KUKA KRL program: UP24.src, Up24.dat

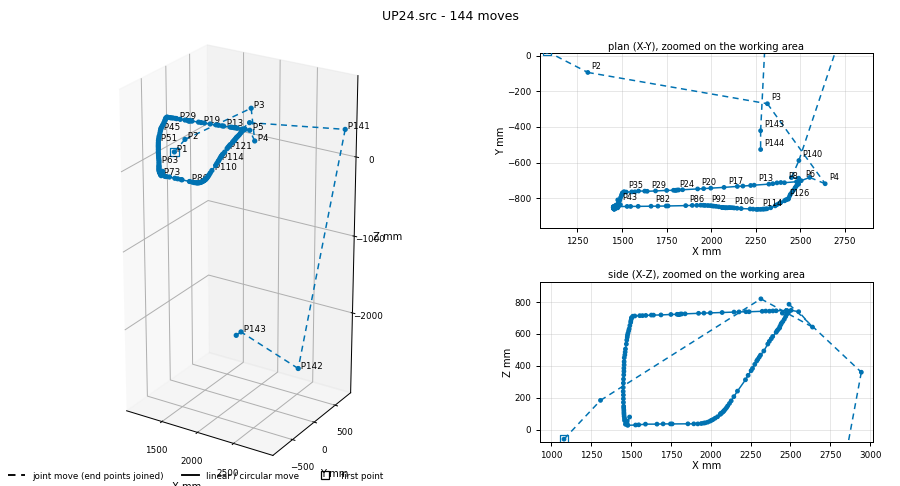
[picture p0: tool path of UP24.src, 144 of 144 moves have a stored position in this frame; points joined in program order, loops and branches not executed]
--- UP24.src ---
&ACCESS RVO1
&REL 1255
&COMMENT VW380 Klebeauftrag_AFO415600
&PARAM EDITMASK = Up999[1-999]
&PARAM TEMPLATE = C:\KRC\Roboter\Template\upvorgabe
&PARAM TPVW_VERSION = 8.3.18
&PARAM DISKPATH = KRC:\R1\UPs
DEF UP24()
   ; FOLD UP Anfang;%{SE} %MKUKATPVW
   SPS_N=-1
   SPS_FERTIG=FALSE
   IF NOT CALLBYSELECT THEN
      INTERRUPT DECL 10 WHEN $CYCFLAG[254]==FALSE DO VW(#FB_STOP,TRUE)
      INTERRUPT ON 10
      INT10=TRUE
      VW_USR_R (#USR_INIT)
   ENDIF
   VW(#VW_INIT_UP,TRUE)
   ; ENDFOLD
   ;FOLD -- VW380, THIL -- ;%{PSE}%MKUKATPVW,%CVW_COM,%VCOMMENT,%P 1:Comment:, 2:VW380, THIL
      ;FOLD {H}
         M_COMMENT("VW380, THIL")
      ;ENDFOLD
   ;ENDFOLD
   ;FOLD -- 415600R01 -- ;%{PSE}%MKUKATPVW,%CVW_COM,%VCOMMENT,%P 1:Comment:, 2:415600R01
      ;FOLD {H}
         M_COMMENT("415600R01")
      ;ENDFOLD
   ;ENDFOLD
   ;FOLD -- FRG ST415600 -- ;%{PSE}%MKUKATPVW,%CVW_COM,%VCOMMENT,%P 1:Comment:, 2:FRG ST415600
      ;FOLD {H}
         M_COMMENT("FRG ST415600")
      ;ENDFOLD
   ;ENDFOLD
   ;FOLD -- ACHTUNG! Position ist nicht von PF0 anfahrbar! -- ;%{PSE}%MKUKATPVW,%CVW_COM,%VCOMMENT,%P 1:Comment:, 2:ACHTUNG! Position ist nicht von PF0 anfahrbar!
      ;FOLD {H}
         M_COMMENT("ACHTUNG! Position ist nicht von PF0 anfahrbar!")
      ;ENDFOLD
   ;ENDFOLD
   ;FOLD PTP VB=100% VE=0% ACC=100% RobWzg=1 Base=2 SPSTrig=0[1/100s] P ;%{P}%MKUKATPVW,%CMOVE8,%VPTP,%P 1:1, 2: VB=, 3:100, 4:%, 5: VE=, 6:0, 7:%, 8: ACC=, 9:100, 10:%, 11: RobWzg=, 12:1, 13: Base=, 14:2, 15: SPSTrig=, 16:0, 17:[1/100s], 18: P, 19:1, 20:-1, 21:200001
      ;FOLD 1: FB PSPS = EIN ;%{SE}%MKUKATPVW %CVW_SPS %VFBPSPS %P 2:FB PSPS = EIN,3:FBPSPS
      ;ENDFOLD
      ;FOLD 2: t5 ( EIN ) = 0[1/10Sek] ;%{SE}%MKUKATPVW %CVW_SPS %VTASG %P 2:t5 ( EIN ) = 0[1/10Sek],3:TASG
      ;ENDFOLD
      ;FOLD 3: A23 = AUS ;%{SE}%MKUKATPVW %CVW_SPS %VBOASG %P 2:A23 = AUS,3:BOASG
      ;ENDFOLD
      ;FOLD 4: SPSMAKRO50 = EIN ;%{SE}%MKUKATPVW %CVW_SPS %VMAKRO %P 2:SPSMAKRO50 = EIN,3:MAKRO
      ;ENDFOLD
      ;FOLD 5: A65 = AUS ;%{SE}%MKUKATPVW %CVW_SPS %VBOASG %P 2:A65 = AUS,3:BOASG
      ;ENDFOLD
      ;FOLD 6: A68 = EIN ;%{SE}%MKUKATPVW %CVW_SPS %VBOASG %P 2:A68 = EIN,3:BOASG
      ;ENDFOLD
      ;FOLD 7: A69 = AUS ;%{SE}%MKUKATPVW %CVW_SPS %VBOASG %P 2:A69 = AUS,3:BOASG
      ;ENDFOLD
      ;FOLD 8: A71 = AUS ;%{SE}%MKUKATPVW %CVW_SPS %VBOASG %P 2:A71 = AUS,3:BOASG
      ;ENDFOLD
      ;FOLD 9: A72 = EIN ;%{SE}%MKUKATPVW %CVW_SPS %VBOASG %P 2:A72 = EIN,3:BOASG
      ;ENDFOLD
      ;FOLD 10: A73 = AUS ;%{SE}%MKUKATPVW %CVW_SPS %VBOASG %P 2:A73 = AUS,3:BOASG
      ;ENDFOLD
      ;FOLD 11: A76 = EIN ;%{SE}%MKUKATPVW %CVW_SPS %VBOASG %P 2:A76 = EIN,3:BOASG
      ;ENDFOLD
      ;FOLD 12: A77 = AUS ;%{SE}%MKUKATPVW %CVW_SPS %VBOASG %P 2:A77 = AUS,3:BOASG
      ;ENDFOLD
      ;FOLD 13: A80 = EIN ;%{SE}%MKUKATPVW %CVW_SPS %VBOASG %P 2:A80 = EIN,3:BOASG
      ;ENDFOLD
      ;FOLD 14: F930 = AUS ;%{SE}%MKUKATPVW %CVW_SPS %VBOASG %P 2:F930 = AUS,3:BOASG
      ;ENDFOLD
      ;FOLD 15: F939 = AUS ;%{SE}%MKUKATPVW %CVW_SPS %VBOASG %P 2:F939 = AUS,3:BOASG
      ;ENDFOLD
      ;FOLD 16: F1 = EIN ;%{SE}%MKUKATPVW %CVW_SPS %VBOASG %P 2:F1 = EIN,3:BOASG
      ;ENDFOLD
      ;FOLD 17: SPSMAKRO343 = !M32 ;%{SE}%MKUKATPVW %CVW_SPS %VMAKRO %P 2:SPSMAKRO343 = !M32,3:MAKRO
      ;ENDFOLD
      ;FOLD 18: SPSMAKRO340 = EIN ;%{SE}%MKUKATPVW %CVW_SPS %VMAKRO %P 2:SPSMAKRO340 = EIN,3:MAKRO
      ;ENDFOLD
      ;FOLD 19: WARTE BIS M13 & M32 ;%{SE}%MKUKATPVW %CVW_SPS %VWBOASG %P 2:WARTE BIS M13 & M32,3:WBOASG
      ;ENDFOLD
      ;FOLD 20: A1521 = EIN ;%{SE}%MKUKATPVW %CVW_SPS %VBOASG %P 2:A1521 = EIN,3:BOASG
      ;ENDFOLD
      ;FOLD 21: A1522 = AUS ;%{SE}%MKUKATPVW %CVW_SPS %VBOASG %P 2:A1522 = AUS,3:BOASG
      ;ENDFOLD
      ;FOLD 22: A1523 = AUS ;%{SE}%MKUKATPVW %CVW_SPS %VBOASG %P 2:A1523 = AUS,3:BOASG
      ;ENDFOLD
      ;FOLD 23: WARTE BIS E1521 & !E1522 & !E1523 ;%{SE}%MKUKATPVW %CVW_SPS %VWBOASG %P 2:WARTE BIS E1521 & !E1522 & !E1523,3:WBOASG
      ;ENDFOLD
      ;FOLD 24: WARTE BIS M13 & M32 ;%{SE}%MKUKATPVW %CVW_SPS %VWBOASG %P 2:WARTE BIS M13 & M32,3:WBOASG
      ;ENDFOLD
      ;FOLD 25: bin10 ( EIN ) = 20 ;%{SE}%MKUKATPVW %CVW_SPS %VARIASG %P 2:bin10 ( EIN ) = 20,3:ARIASG
      ;ENDFOLD
      ;FOLD 26: bin11 ( EIN ) = 1 ;%{SE}%MKUKATPVW %CVW_SPS %VARIASG %P 2:bin11 ( EIN ) = 1,3:ARIASG
      ;ENDFOLD
      ;FOLD 27: F341 = EIN ;%{SE}%MKUKATPVW %CVW_SPS %VBOASG %P 2:F341 = EIN,3:BOASG
      ;ENDFOLD
      ;FOLD 28: ana1 ( EIN ) = VPROP: 500 [mm/Sek] OFFS: 0[mV] DELAY:0 [ms] ;%{SE}%MKUKATPVW %CVW_SPS %VANAVPROP %P 2:ana1 ( EIN ) = VPROP: 500 [mm/Sek] OFFS: 0[mV] DELAY:0 [ms],3:ANAVPROP
      ;ENDFOLD
      ;FOLD 29: A43 = AUS ;%{SE}%MKUKATPVW %CVW_SPS %VBOASG %P 2:A43 = AUS,3:BOASG
      ;ENDFOLD
      ;FOLD 30: A44 = AUS ;%{SE}%MKUKATPVW %CVW_SPS %VBOASG %P 2:A44 = AUS,3:BOASG
      ;ENDFOLD
      ;FOLD 31: WARTE BIS M32 & M34 & E43 & E44 & E63 & E71 ;%{SE}%MKUKATPVW %CVW_SPS %VWBOASG %P 2:WARTE BIS M32 & M34 & E43 & E44 & E63 & E71,3:WBOASG
      ;ENDFOLD
      ;FOLD 32: WARTE BIS E23 ;%{SE}%MKUKATPVW %CVW_SPS %VWBOASG %P 2:WARTE BIS E23,3:WBOASG
      ;ENDFOLD
      ;FOLD 33: A23 = EIN ;%{SE}%MKUKATPVW %CVW_SPS %VBOASG %P 2:A23 = EIN,3:BOASG
      ;ENDFOLD
      ;FOLD 34: FB PSPS = M13 & M30 & M32 & M34 & E43 & E44 & E63 & E71 ;%{SE}%MKUKATPVW %CVW_SPS %VFBPSPS %P 2:FB PSPS = M13 & M30 & M32 & M34 & E43 & E44 & E63 & E71,3:FBPSPS
      ;ENDFOLD
      ;FOLD {H}
         VW_MPARA_ACT=P1_D
         Act_P1 = P1
         Act_P2 = P1
         VW(#MPARA,TRUE)
         SPS_FERTIG=FALSE
         SPS_FERTIG_ANA=FALSE
         TRIGGER WHEN DISTANCE=1 DELAY=0 DO SPS_TRIG(1) PRIO=-1
         TRIGGER WHEN DISTANCE=1 DELAY=0 DO SPS_TRIG(20002) PRIO=-1
         PTP P1
         $ADVANCE=1
         WAIT FOR SPS_FERTIG
         WAIT FOR SPS_FERTIG_ANA
      ;ENDFOLD
   ;ENDFOLD
   ;FOLD PTP VB=100% VE=100% ACC=100% RobWzg=1 Base=2 SPSTrig=0[1/100s] P ;%{P}%MKUKATPVW,%CMOVE8,%VPTP,%P 1:1, 2: VB=, 3:100, 4:%, 5: VE=, 6:100, 7:%, 8: ACC=, 9:100, 10:%, 11: RobWzg=, 12:1, 13: Base=, 14:2, 15: SPSTrig=, 16:0, 17:[1/100s], 18: P, 19:2, 20:-1, 21:3
      ;FOLD 1: FB PSPS = M13 & M30 & M32 & M34 & E43 & E44 & E63 & E71 ;%{SE}%MKUKATPVW %CVW_SPS %VFBPSPS %P 2:FB PSPS = M13 & M30 & M32 & M34 & E43 & E44 & E63 & E71,3:FBPSPS
      ;ENDFOLD
      ;FOLD {H}
         VW_MPARA_ACT=P2_D
         Act_P1 = P2
         Act_P2 = P2
         VW(#MPARA,TRUE)
         SPS_FERTIG=FALSE
         TRIGGER WHEN DISTANCE=1 DELAY=0 DO SPS_TRIG(10003) PRIO=-1 UP_TIME_OUT=SPS_TIMEOUT
         PTP P2 C_PTP C_VEL
         $ADVANCE=1
      ;ENDFOLD
   ;ENDFOLD
   ;FOLD PTP VB=100% VE=100% ACC=100% RobWzg=1 Base=2 SPSTrig=0[1/100s] P ;%{P}%MKUKATPVW,%CMOVE8,%VPTP,%P 1:1, 2: VB=, 3:100, 4:%, 5: VE=, 6:100, 7:%, 8: ACC=, 9:100, 10:%, 11: RobWzg=, 12:1, 13: Base=, 14:2, 15: SPSTrig=, 16:0, 17:[1/100s], 18: P, 19:3, 20:-1, 21:4
      ;FOLD 1: FB PSPS = M13 & M30 & M32 & M34 & E43 & E44 & E63 & E71 ;%{SE}%MKUKATPVW %CVW_SPS %VFBPSPS %P 2:FB PSPS = M13 & M30 & M32 & M34 & E43 & E44 & E63 & E71,3:FBPSPS
      ;ENDFOLD
      ;FOLD {H}
         VW_MPARA_ACT=P3_D
         Act_P1 = P3
         Act_P2 = P3
         VW(#MPARA,TRUE)
         SPS_FERTIG=FALSE
         TRIGGER WHEN DISTANCE=1 DELAY=0 DO SPS_TRIG(10004) PRIO=-1 UP_TIME_OUT=SPS_TIMEOUT
         PTP P3 C_PTP C_VEL
         $ADVANCE=1
      ;ENDFOLD
   ;ENDFOLD
   ;FOLD PTP VB=100% VE=100% ACC=100% RobWzg=1 Base=2 SPSTrig=0[1/100s] P ;%{P}%MKUKATPVW,%CMOVE8,%VPTP,%P 1:1, 2: VB=, 3:100, 4:%, 5: VE=, 6:100, 7:%, 8: ACC=, 9:100, 10:%, 11: RobWzg=, 12:1, 13: Base=, 14:2, 15: SPSTrig=, 16:0, 17:[1/100s], 18: P, 19:4, 20:-1, 21:5
      ;FOLD 1: FB PSPS = M13 & M30 & M32 & M34 & E43 & E44 & E63 & E71 ;%{SE}%MKUKATPVW %CVW_SPS %VFBPSPS %P 2:FB PSPS = M13 & M30 & M32 & M34 & E43 & E44 & E63 & E71,3:FBPSPS
      ;ENDFOLD
      ;FOLD {H}
         VW_MPARA_ACT=P4_D
         Act_P1 = P4
         Act_P2 = P4
         VW(#MPARA,TRUE)
         SPS_FERTIG=FALSE
         TRIGGER WHEN DISTANCE=1 DELAY=0 DO SPS_TRIG(10005) PRIO=-1 UP_TIME_OUT=SPS_TIMEOUT
         PTP P4 C_PTP C_VEL
         $ADVANCE=1
      ;ENDFOLD
   ;ENDFOLD
   ;FOLD PTP VB=100% VE=0% ACC=100% RobWzg=1 Base=2 SPSTrig=0[1/100s] P ;%{P}%MKUKATPVW,%CMOVE8,%VPTP,%P 1:1, 2: VB=, 3:100, 4:%, 5: VE=, 6:0, 7:%, 8: ACC=, 9:100, 10:%, 11: RobWzg=, 12:1, 13: Base=, 14:2, 15: SPSTrig=, 16:0, 17:[1/100s], 18: P, 19:5, 20:-1, 21:6
      ;FOLD 1: FB PSPS = EIN ;%{SE}%MKUKATPVW %CVW_SPS %VFBPSPS %P 2:FB PSPS = EIN,3:FBPSPS
      ;ENDFOLD
      ;FOLD 2: A23 = AUS ;%{SE}%MKUKATPVW %CVW_SPS %VBOASG %P 2:A23 = AUS,3:BOASG
      ;ENDFOLD
      ;FOLD 3: SPSMAKRO182 = E1534 + E163 ;%{SE}%MKUKATPVW %CVW_SPS %VMAKRO %P 2:SPSMAKRO182 = E1534 + E163,3:MAKRO
      ;ENDFOLD
      ;FOLD 4: SPSMAKRO183 = !E15 ;%{SE}%MKUKATPVW %CVW_SPS %VMAKRO %P 2:SPSMAKRO183 = !E15,3:MAKRO
      ;ENDFOLD
      ;FOLD 5: WARTE BIS !E1534 & !E1535 ;%{SE}%MKUKATPVW %CVW_SPS %VWBOASG %P 2:WARTE BIS !E1534 & !E1535,3:WBOASG
      ;ENDFOLD
      ;FOLD 6: SPSMAKRO180 = !E15 ;%{SE}%MKUKATPVW %CVW_SPS %VMAKRO %P 2:SPSMAKRO180 = !E15,3:MAKRO
      ;ENDFOLD
      ;FOLD 7: WARTE BIS E23 ;%{SE}%MKUKATPVW %CVW_SPS %VWBOASG %P 2:WARTE BIS E23,3:WBOASG
      ;ENDFOLD
      ;FOLD 8: A23 = EIN ;%{SE}%MKUKATPVW %CVW_SPS %VBOASG %P 2:A23 = EIN,3:BOASG
      ;ENDFOLD
      ;FOLD 9: FB PSPS = M13 & M30 & M32 & M34 & E43 & E44 & E63 & E71 ;%{SE}%MKUKATPVW %CVW_SPS %VFBPSPS %P 2:FB PSPS = M13 & M30 & M32 & M34 & E43 & E44 & E63 & E71,3:FBPSPS
      ;ENDFOLD
      ;FOLD {H}
         VW_MPARA_ACT=P5_D
         Act_P1 = P5
         Act_P2 = P5
         VW(#MPARA,TRUE)
         SPS_FERTIG=FALSE
         TRIGGER WHEN DISTANCE=1 DELAY=0 DO SPS_TRIG(6) PRIO=-1
         PTP P5
         $ADVANCE=1
         WAIT FOR SPS_FERTIG
      ;ENDFOLD
   ;ENDFOLD
   ;FOLD -- ACHTUNG! BEI KLEBEN START UNBEDINGT SATZ 5 ANWAEHLEN -- ;%{PSE}%MKUKATPVW,%CVW_COM,%VCOMMENT,%P 1:Comment:, 2:ACHTUNG! BEI KLEBEN START UNBEDINGT SATZ 5 ANWAEHLEN
      ;FOLD {H}
         M_COMMENT("ACHTUNG! BEI KLEBEN START UNBEDINGT SATZ 5 ANWAEHLEN")
      ;ENDFOLD
   ;ENDFOLD
   ;FOLD KLIN VB=150[mm/s] Genau=30[mm] ACC=50% RobWzg=1 Base=2 SPSTrig=0[1/100s] P ;%{P}%MKUKATPVW,%CMOVE8,%VKLIN,%P 1:4, 2: VB=, 3:150, 4:[mm/s], 5: Genau=, 6:30, 7:[mm], 8: ACC=, 9:50, 10:%, 11: RobWzg=, 12:1, 13: Base=, 14:2, 15: SPSTrig=, 16:0, 17:[1/100s], 18: P, 19:6, 20:-1, 21:7
      ;FOLD 1: FB PSPS = M13 & M30 & M32 & M34 & E43 & E44 & E63 & E71 ;%{SE}%MKUKATPVW %CVW_SPS %VFBPSPS %P 2:FB PSPS = M13 & M30 & M32 & M34 & E43 & E44 & E63 & E71,3:FBPSPS
      ;ENDFOLD
      ;FOLD {H}
         VW_MPARA_ACT=P6_D
         Act_P1 = P6
         Act_P2 = P6
         VW(#MPARA,TRUE)
         SPS_FERTIG=FALSE
         TRIGGER WHEN DISTANCE=1 DELAY=0 DO SPS_TRIG(10007) PRIO=-1 UP_TIME_OUT=SPS_TIMEOUT
         LIN P6 C_DIS
         $ADVANCE=1
      ;ENDFOLD
   ;ENDFOLD
   ;FOLD -- Start Klebenaht 5H4_833_055_C0006_A__1150_000100_LL -- ;%{PSE}%MKUKATPVW,%CVW_COM,%VCOMMENT,%P 1:Comment:, 2:Start Klebenaht 5H4_833_055_C0006_A__1150_000100_LL
      ;FOLD {H}
         M_COMMENT("Start Klebenaht 5H4_833_055_C0006_A__1150_000100_LL")
      ;ENDFOLD
   ;ENDFOLD
   ;FOLD -- Schaltpunkt 1 -- ;%{PSE}%MKUKATPVW,%CVW_COM,%VCOMMENT,%P 1:Comment:, 2:Schaltpunkt 1
      ;FOLD {H}
         M_COMMENT("Schaltpunkt 1")
      ;ENDFOLD
   ;ENDFOLD
   ;FOLD KLIN VB=150[mm/s] Genau=30[mm] ACC=50% RobWzg=1 Base=2 SPSTrig=5[1/100s] P ;%{P}%MKUKATPVW,%CMOVE8,%VKLIN,%P 1:4, 2: VB=, 3:150, 4:[mm/s], 5: Genau=, 6:30, 7:[mm], 8: ACC=, 9:50, 10:%, 11: RobWzg=, 12:1, 13: Base=, 14:2, 15: SPSTrig=, 16:5, 17:[1/100s], 18: P, 19:7, 20:-1, 21:8
      ;FOLD BS A1544 ( EIN ) = !E15 Schaltpkt:2[mm]:-50[ms] ;%{SE}%MKUKATPVW %CVW_SPS %VBSBO %P 2:BS A1544 ( EIN ) = !E15 Schaltpkt:2[mm]:-50[ms],3:BSBO
      ;ENDFOLD
      ;FOLD 1: FB PSPS = M13 & M30 & M32 & M34 & E43 & E44 & E63 & E71 ;%{SE}%MKUKATPVW %CVW_SPS %VFBPSPS %P 2:FB PSPS = M13 & M30 & M32 & M34 & E43 & E44 & E63 & E71,3:FBPSPS
      ;ENDFOLD
      ;FOLD {H}
         VW_MPARA_ACT=P7_D
         Act_P1 = P7
         Act_P2 = P7
         VW(#MPARA,TRUE)
         SPS_FERTIG=FALSE
         TRIGGER WHEN DISTANCE=1 DELAY=-50 DO SPS_TRIG(10008) PRIO=-1 UP_TIME_OUT=SPS_TIMEOUT
         TRIGGER WHEN PATH=2 DELAY=-50 DO $OUT[1544]=(NOT $IN[15])
         LIN P7 C_DIS
         $ADVANCE=1
      ;ENDFOLD
   ;ENDFOLD
   ;FOLD -- Ende Klebenaht 5H4_833_055_C0006_A__1150_000100_LL -- ;%{PSE}%MKUKATPVW,%CVW_COM,%VCOMMENT,%P 1:Comment:, 2:Ende Klebenaht 5H4_833_055_C0006_A__1150_000100_LL
      ;FOLD {H}
         M_COMMENT("Ende Klebenaht 5H4_833_055_C0006_A__1150_000100_LL")
      ;ENDFOLD
   ;ENDFOLD
   ;FOLD -- Schaltpunkt 2 -- ;%{PSE}%MKUKATPVW,%CVW_COM,%VCOMMENT,%P 1:Comment:, 2:Schaltpunkt 2
      ;FOLD {H}
         M_COMMENT("Schaltpunkt 2")
      ;ENDFOLD
   ;ENDFOLD
   ;FOLD KLIN VB=150[mm/s] Genau=30[mm] ACC=50% RobWzg=1 Base=2 SPSTrig=5[1/100s] P ;%{P}%MKUKATPVW,%CMOVE8,%VKLIN,%P 1:4, 2: VB=, 3:150, 4:[mm/s], 5: Genau=, 6:30, 7:[mm], 8: ACC=, 9:50, 10:%, 11: RobWzg=, 12:1, 13: Base=, 14:2, 15: SPSTrig=, 16:5, 17:[1/100s], 18: P, 19:8, 20:-1, 21:9
      ;FOLD BS A1544 ( EIN ) = AUS Schaltpkt:-1[mm]:-50[ms] ;%{SE}%MKUKATPVW %CVW_SPS %VBSBO %P 2:BS A1544 ( EIN ) = AUS Schaltpkt:-1[mm]:-50[ms],3:BSBO
      ;ENDFOLD
      ;FOLD BS bin11 ( EIN ) = 2 Schaltpkt:5[mm]:-50[ms] ;%{SE}%MKUKATPVW %CVW_SPS %VBSARI %P 2:BS bin11 ( EIN ) = 2 Schaltpkt:5[mm]:-50[ms],3:BSARI
      ;ENDFOLD
      ;FOLD 1: FB PSPS = M13 & M30 & M32 & M34 & E43 & E44 & E63 & E71 ;%{SE}%MKUKATPVW %CVW_SPS %VFBPSPS %P 2:FB PSPS = M13 & M30 & M32 & M34 & E43 & E44 & E63 & E71,3:FBPSPS
      ;ENDFOLD
      ;FOLD {H}
         VW_MPARA_ACT=P8_D
         Act_P1 = P8
         Act_P2 = P8
         VW(#MPARA,TRUE)
         SPS_FERTIG=FALSE
         TRIGGER WHEN DISTANCE=1 DELAY=-50 DO SPS_TRIG(10009) PRIO=-1 UP_TIME_OUT=SPS_TIMEOUT
         TRIGGER WHEN PATH=-1 DELAY=-50 DO $OUT[1544]=(FALSE)
         TRIGGER WHEN PATH=5 DELAY=-50 DO $B_OUT[11]=(2)
         LIN P8 C_DIS
         $ADVANCE=1
      ;ENDFOLD
   ;ENDFOLD
   ;FOLD KLIN VB=150[mm/s] Genau=30[mm] ACC=50% RobWzg=1 Base=2 SPSTrig=0[1/100s] P ;%{P}%MKUKATPVW,%CMOVE8,%VKLIN,%P 1:4, 2: VB=, 3:150, 4:[mm/s], 5: Genau=, 6:30, 7:[mm], 8: ACC=, 9:50, 10:%, 11: RobWzg=, 12:1, 13: Base=, 14:2, 15: SPSTrig=, 16:0, 17:[1/100s], 18: P, 19:9, 20:-1, 21:10
      ;FOLD 1: FB PSPS = M13 & M30 & M32 & M34 & E43 & E44 & E63 & E71 ;%{SE}%MKUKATPVW %CVW_SPS %VFBPSPS %P 2:FB PSPS = M13 & M30 & M32 & M34 & E43 & E44 & E63 & E71,3:FBPSPS
      ;ENDFOLD
      ;FOLD {H}
         VW_MPARA_ACT=P9_D
         Act_P1 = P9
         Act_P2 = P9
         VW(#MPARA,TRUE)
         SPS_FERTIG=FALSE
         TRIGGER WHEN DISTANCE=1 DELAY=0 DO SPS_TRIG(10010) PRIO=-1 UP_TIME_OUT=SPS_TIMEOUT
         LIN P9 C_DIS
         $ADVANCE=1
      ;ENDFOLD
   ;ENDFOLD
   ;FOLD KLIN VB=200[mm/s] Genau=40[mm] ACC=50% RobWzg=1 Base=2 SPSTrig=0[1/100s] P ;%{P}%MKUKATPVW,%CMOVE8,%VKLIN,%P 1:4, 2: VB=, 3:200, 4:[mm/s], 5: Genau=, 6:40, 7:[mm], 8: ACC=, 9:50, 10:%, 11: RobWzg=, 12:1, 13: Base=, 14:2, 15: SPSTrig=, 16:0, 17:[1/100s], 18: P, 19:10, 20:-1, 21:11
      ;FOLD 1: FB PSPS = M13 & M30 & M32 & M34 & E43 & E44 & E63 & E71 ;%{SE}%MKUKATPVW %CVW_SPS %VFBPSPS %P 2:FB PSPS = M13 & M30 & M32 & M34 & E43 & E44 & E63 & E71,3:FBPSPS
      ;ENDFOLD
      ;FOLD {H}
         VW_MPARA_ACT=P10_D
         Act_P1 = P10
         Act_P2 = P10
         VW(#MPARA,TRUE)
         SPS_FERTIG=FALSE
         TRIGGER WHEN DISTANCE=1 DELAY=0 DO SPS_TRIG(10011) PRIO=-1 UP_TIME_OUT=SPS_TIMEOUT
         LIN P10 C_DIS
         $ADVANCE=1
      ;ENDFOLD
   ;ENDFOLD
   ;FOLD -- Start Klebenaht 5H4_833_055_C0002_A__1110_000100_LL -- ;%{PSE}%MKUKATPVW,%CVW_COM,%VCOMMENT,%P 1:Comment:, 2:Start Klebenaht 5H4_833_055_C0002_A__1110_000100_LL
      ;FOLD {H}
         M_COMMENT("Start Klebenaht 5H4_833_055_C0002_A__1110_000100_LL")
      ;ENDFOLD
   ;ENDFOLD
   ;FOLD KLIN VB=200[mm/s] Genau=40[mm] ACC=50% RobWzg=1 Base=2 SPSTrig=5[1/100s] P ;%{P}%MKUKATPVW,%CMOVE8,%VKLIN,%P 1:4, 2: VB=, 3:200, 4:[mm/s], 5: Genau=, 6:40, 7:[mm], 8: ACC=, 9:50, 10:%, 11: RobWzg=, 12:1, 13: Base=, 14:2, 15: SPSTrig=, 16:5, 17:[1/100s], 18: P, 19:11, 20:-1, 21:12
      ;FOLD BS A1544 ( EIN ) = !E15 Schaltpkt:2[mm]:-50[ms] ;%{SE}%MKUKATPVW %CVW_SPS %VBSBO %P 2:BS A1544 ( EIN ) = !E15 Schaltpkt:2[mm]:-50[ms],3:BSBO
      ;ENDFOLD
      ;FOLD 1: FB PSPS = M13 & M30 & M32 & M34 & E43 & E44 & E63 & E71 ;%{SE}%MKUKATPVW %CVW_SPS %VFBPSPS %P 2:FB PSPS = M13 & M30 & M32 & M34 & E43 & E44 & E63 & E71,3:FBPSPS
      ;ENDFOLD
      ;FOLD {H}
         VW_MPARA_ACT=P11_D
         Act_P1 = P11
         Act_P2 = P11
         VW(#MPARA,TRUE)
         SPS_FERTIG=FALSE
         TRIGGER WHEN DISTANCE=1 DELAY=-50 DO SPS_TRIG(10012) PRIO=-1 UP_TIME_OUT=SPS_TIMEOUT
         TRIGGER WHEN PATH=2 DELAY=-50 DO $OUT[1544]=(NOT $IN[15])
         LIN P11 C_DIS
         $ADVANCE=1
      ;ENDFOLD
   ;ENDFOLD
   ;FOLD KLIN VB=200[mm/s] Genau=40[mm] ACC=50% RobWzg=1 Base=2 SPSTrig=0[1/100s] P ;%{P}%MKUKATPVW,%CMOVE8,%VKLIN,%P 1:4, 2: VB=, 3:200, 4:[mm/s], 5: Genau=, 6:40, 7:[mm], 8: ACC=, 9:50, 10:%, 11: RobWzg=, 12:1, 13: Base=, 14:2, 15: SPSTrig=, 16:0, 17:[1/100s], 18: P, 19:12, 20:-1, 21:13
      ;FOLD 1: FB PSPS = M13 & M30 & M32 & M34 & E43 & E44 & E63 & E71 ;%{SE}%MKUKATPVW %CVW_SPS %VFBPSPS %P 2:FB PSPS = M13 & M30 & M32 & M34 & E43 & E44 & E63 & E71,3:FBPSPS
      ;ENDFOLD
      ;FOLD {H}
         VW_MPARA_ACT=P12_D
         Act_P1 = P12
         Act_P2 = P12
         VW(#MPARA,TRUE)
         SPS_FERTIG=FALSE
         TRIGGER WHEN DISTANCE=1 DELAY=0 DO SPS_TRIG(10013) PRIO=-1 UP_TIME_OUT=SPS_TIMEOUT
         LIN P12 C_DIS
         $ADVANCE=1
      ;ENDFOLD
   ;ENDFOLD
   ;FOLD -- Schaltpunkt 3 -- ;%{PSE}%MKUKATPVW,%CVW_COM,%VCOMMENT,%P 1:Comment:, 2:Schaltpunkt 3
      ;FOLD {H}
         M_COMMENT("Schaltpunkt 3")
      ;ENDFOLD
   ;ENDFOLD
   ;FOLD KLIN VB=200[mm/s] Genau=40[mm] ACC=50% RobWzg=1 Base=2 SPSTrig=5[1/100s] P ;%{P}%MKUKATPVW,%CMOVE8,%VKLIN,%P 1:4, 2: VB=, 3:200, 4:[mm/s], 5: Genau=, 6:40, 7:[mm], 8: ACC=, 9:50, 10:%, 11: RobWzg=, 12:1, 13: Base=, 14:2, 15: SPSTrig=, 16:5, 17:[1/100s], 18: P, 19:13, 20:-1, 21:14
      ;FOLD BS bin11 ( EIN ) = 3 Schaltpkt:5[mm]:-50[ms] ;%{SE}%MKUKATPVW %CVW_SPS %VBSARI %P 2:BS bin11 ( EIN ) = 3 Schaltpkt:5[mm]:-50[ms],3:BSARI
      ;ENDFOLD
      ;FOLD 1: FB PSPS = M13 & M30 & M32 & M34 & E43 & E44 & E63 & E71 ;%{SE}%MKUKATPVW %CVW_SPS %VFBPSPS %P 2:FB PSPS = M13 & M30 & M32 & M34 & E43 & E44 & E63 & E71,3:FBPSPS
      ;ENDFOLD
      ;FOLD {H}
         VW_MPARA_ACT=P13_D
         Act_P1 = P13
         Act_P2 = P13
         VW(#MPARA,TRUE)
         SPS_FERTIG=FALSE
         TRIGGER WHEN DISTANCE=1 DELAY=-50 DO SPS_TRIG(10014) PRIO=-1 UP_TIME_OUT=SPS_TIMEOUT
         TRIGGER WHEN PATH=5 DELAY=-50 DO $B_OUT[11]=(3)
         LIN P13 C_DIS
         $ADVANCE=1
      ;ENDFOLD
   ;ENDFOLD
   ;FOLD KLIN VB=200[mm/s] Genau=40[mm] ACC=50% RobWzg=1 Base=2 SPSTrig=0[1/100s] P ;%{P}%MKUKATPVW,%CMOVE8,%VKLIN,%P 1:4, 2: VB=, 3:200, 4:[mm/s], 5: Genau=, 6:40, 7:[mm], 8: ACC=, 9:50, 10:%, 11: RobWzg=, 12:1, 13: Base=, 14:2, 15: SPSTrig=, 16:0, 17:[1/100s], 18: P, 19:14, 20:-1, 21:15
      ;FOLD 1: FB PSPS = M13 & M30 & M32 & M34 & E43 & E44 & E63 & E71 ;%{SE}%MKUKATPVW %CVW_SPS %VFBPSPS %P 2:FB PSPS = M13 & M30 & M32 & M34 & E43 & E44 & E63 & E71,3:FBPSPS
      ;ENDFOLD
      ;FOLD {H}
         VW_MPARA_ACT=P14_D
         Act_P1 = P14
         Act_P2 = P14
         VW(#MPARA,TRUE)
         SPS_FERTIG=FALSE
         TRIGGER WHEN DISTANCE=1 DELAY=0 DO SPS_TRIG(10015) PRIO=-1 UP_TIME_OUT=SPS_TIMEOUT
         LIN P14 C_DIS
         $ADVANCE=1
      ;ENDFOLD
   ;ENDFOLD
   ;FOLD -- Schaltpunkt 4 -- ;%{PSE}%MKUKATPVW,%CVW_COM,%VCOMMENT,%P 1:Comment:, 2:Schaltpunkt 4
      ;FOLD {H}
         M_COMMENT("Schaltpunkt 4")
      ;ENDFOLD
   ;ENDFOLD
   ;FOLD KLIN VB=200[mm/s] Genau=40[mm] ACC=50% RobWzg=1 Base=2 SPSTrig=0[1/100s] P ;%{P}%MKUKATPVW,%CMOVE8,%VKLIN,%P 1:4, 2: VB=, 3:200, 4:[mm/s], 5: Genau=, 6:40, 7:[mm], 8: ACC=, 9:50, 10:%, 11: RobWzg=, 12:1, 13: Base=, 14:2, 15: SPSTrig=, 16:0, 17:[1/100s], 18: P, 19:15, 20:-1, 21:16
      ;FOLD BS bin11 ( EIN ) = 4 Schaltpkt:5[mm]:-50[ms] ;%{SE}%MKUKATPVW %CVW_SPS %VBSARI %P 2:BS bin11 ( EIN ) = 4 Schaltpkt:5[mm]:-50[ms],3:BSARI
      ;ENDFOLD
      ;FOLD 1: FB PSPS = M13 & M30 & M32 & M34 & E43 & E44 & E63 & E71 ;%{SE}%MKUKATPVW %CVW_SPS %VFBPSPS %P 2:FB PSPS = M13 & M30 & M32 & M34 & E43 & E44 & E63 & E71,3:FBPSPS
      ;ENDFOLD
      ;FOLD {H}
         VW_MPARA_ACT=P15_D
         Act_P1 = P15
         Act_P2 = P15
         VW(#MPARA,TRUE)
         SPS_FERTIG=FALSE
         TRIGGER WHEN DISTANCE=1 DELAY=0 DO SPS_TRIG(10016) PRIO=-1 UP_TIME_OUT=SPS_TIMEOUT
         TRIGGER WHEN PATH=5 DELAY=-50 DO $B_OUT[11]=(4)
         LIN P15 C_DIS
         $ADVANCE=1
      ;ENDFOLD
   ;ENDFOLD
   ;FOLD KLIN VB=200[mm/s] Genau=40[mm] ACC=50% RobWzg=1 Base=2 SPSTrig=0[1/100s] P ;%{P}%MKUKATPVW,%CMOVE8,%VKLIN,%P 1:4, 2: VB=, 3:200, 4:[mm/s], 5: Genau=, 6:40, 7:[mm], 8: ACC=, 9:50, 10:%, 11: RobWzg=, 12:1, 13: Base=, 14:2, 15: SPSTrig=, 16:0, 17:[1/100s], 18: P, 19:16, 20:-1, 21:17
      ;FOLD 1: FB PSPS = M13 & M30 & M32 & M34 & E43 & E44 & E63 & E71 ;%{SE}%MKUKATPVW %CVW_SPS %VFBPSPS %P 2:FB PSPS = M13 & M30 & M32 & M34 & E43 & E44 & E63 & E71,3:FBPSPS
      ;ENDFOLD
      ;FOLD {H}
         VW_MPARA_ACT=P16_D
         Act_P1 = P16
         Act_P2 = P16
         VW(#MPARA,TRUE)
         SPS_FERTIG=FALSE
         TRIGGER WHEN DISTANCE=1 DELAY=0 DO SPS_TRIG(10017) PRIO=-1 UP_TIME_OUT=SPS_TIMEOUT
         LIN P16 C_DIS
         $ADVANCE=1
      ;ENDFOLD
   ;ENDFOLD
   ;FOLD KLIN VB=200[mm/s] Genau=40[mm] ACC=50% RobWzg=1 Base=2 SPSTrig=0[1/100s] P ;%{P}%MKUKATPVW,%CMOVE8,%VKLIN,%P 1:4, 2: VB=, 3:200, 4:[mm/s], 5: Genau=, 6:40, 7:[mm], 8: ACC=, 9:50, 10:%, 11: RobWzg=, 12:1, 13: Base=, 14:2, 15: SPSTrig=, 16:0, 17:[1/100s], 18: P, 19:17, 20:-1, 21:18
      ;FOLD 1: FB PSPS = M13 & M30 & M32 & M34 & E43 & E44 & E63 & E71 ;%{SE}%MKUKATPVW %CVW_SPS %VFBPSPS %P 2:FB PSPS = M13 & M30 & M32 & M34 & E43 & E44 & E63 & E71,3:FBPSPS
      ;ENDFOLD
      ;FOLD {H}
         VW_MPARA_ACT=P17_D
         Act_P1 = P17
         Act_P2 = P17
         VW(#MPARA,TRUE)
         SPS_FERTIG=FALSE
         TRIGGER WHEN DISTANCE=1 DELAY=0 DO SPS_TRIG(10018) PRIO=-1 UP_TIME_OUT=SPS_TIMEOUT
         LIN P17 C_DIS
         $ADVANCE=1
      ;ENDFOLD
   ;ENDFOLD
   ;FOLD -- Schaltpunkt 5 -- ;%{PSE}%MKUKATPVW,%CVW_COM,%VCOMMENT,%P 1:Comment:, 2:Schaltpunkt 5
      ;FOLD {H}
         M_COMMENT("Schaltpunkt 5")
      ;ENDFOLD
   ;ENDFOLD
   ;FOLD -- Vordrucktrigger -- ;%{PSE}%MKUKATPVW,%CVW_COM,%VCOMMENT,%P 1:Comment:, 2:Vordrucktrigger
      ;FOLD {H}
         M_COMMENT("Vordrucktrigger")
      ;ENDFOLD
   ;ENDFOLD
   ;FOLD KLIN VB=200[mm/s] Genau=40[mm] ACC=50% RobWzg=1 Base=2 SPSTrig=0[1/100s] P ;%{P}%MKUKATPVW,%CMOVE8,%VKLIN,%P 1:4, 2: VB=, 3:200, 4:[mm/s], 5: Genau=, 6:40, 7:[mm], 8: ACC=, 9:50, 10:%, 11: RobWzg=, 12:1, 13: Base=, 14:2, 15: SPSTrig=, 16:0, 17:[1/100s], 18: P, 19:18, 20:-1, 21:19
      ;FOLD BS bin11 ( EIN ) = 5 Schaltpkt:5[mm]:-50[ms] ;%{SE}%MKUKATPVW %CVW_SPS %VBSARI %P 2:BS bin11 ( EIN ) = 5 Schaltpkt:5[mm]:-50[ms],3:BSARI
      ;ENDFOLD
      ;FOLD 1: Puls A1533 = Pegel:EIN Zeit:10 [1/10Sek] ;%{SE}%MKUKATPVW %CVW_SPS %VPULS %P 2:Puls A1533 = Pegel:EIN Zeit:10 [1/10Sek],3:PULS
      ;ENDFOLD
      ;FOLD 2: FB PSPS = M13 & M30 & M32 & M34 & E43 & E44 & E63 & E71 ;%{SE}%MKUKATPVW %CVW_SPS %VFBPSPS %P 2:FB PSPS = M13 & M30 & M32 & M34 & E43 & E44 & E63 & E71,3:FBPSPS
      ;ENDFOLD
      ;FOLD {H}
         VW_MPARA_ACT=P18_D
         Act_P1 = P18
         Act_P2 = P18
         VW(#MPARA,TRUE)
         SPS_FERTIG=FALSE
         TRIGGER WHEN DISTANCE=1 DELAY=0 DO SPS_TRIG(10019) PRIO=-1 UP_TIME_OUT=SPS_TIMEOUT
         TRIGGER WHEN PATH=5 DELAY=-50 DO $B_OUT[11]=(5)
         LIN P18 C_DIS
         $ADVANCE=1
      ;ENDFOLD
   ;ENDFOLD
   ;FOLD KLIN VB=200[mm/s] Genau=40[mm] ACC=50% RobWzg=1 Base=2 SPSTrig=0[1/100s] P ;%{P}%MKUKATPVW,%CMOVE8,%VKLIN,%P 1:4, 2: VB=, 3:200, 4:[mm/s], 5: Genau=, 6:40, 7:[mm], 8: ACC=, 9:50, 10:%, 11: RobWzg=, 12:1, 13: Base=, 14:2, 15: SPSTrig=, 16:0, 17:[1/100s], 18: P, 19:19, 20:-1, 21:20
      ;FOLD 1: FB PSPS = M13 & M30 & M32 & M34 & E43 & E44 & E63 & E71 ;%{SE}%MKUKATPVW %CVW_SPS %VFBPSPS %P 2:FB PSPS = M13 & M30 & M32 & M34 & E43 & E44 & E63 & E71,3:FBPSPS
      ;ENDFOLD
      ;FOLD {H}
         VW_MPARA_ACT=P19_D
         Act_P1 = P19
         Act_P2 = P19
         VW(#MPARA,TRUE)
         SPS_FERTIG=FALSE
         TRIGGER WHEN DISTANCE=1 DELAY=0 DO SPS_TRIG(10020) PRIO=-1 UP_TIME_OUT=SPS_TIMEOUT
         LIN P19 C_DIS
         $ADVANCE=1
      ;ENDFOLD
   ;ENDFOLD
   ;FOLD KLIN VB=200[mm/s] Genau=40[mm] ACC=50% RobWzg=1 Base=2 SPSTrig=0[1/100s] P ;%{P}%MKUKATPVW,%CMOVE8,%VKLIN,%P 1:4, 2: VB=, 3:200, 4:[mm/s], 5: Genau=, 6:40, 7:[mm], 8: ACC=, 9:50, 10:%, 11: RobWzg=, 12:1, 13: Base=, 14:2, 15: SPSTrig=, 16:0, 17:[1/100s], 18: P, 19:20, 20:-1, 21:21
      ;FOLD 1: FB PSPS = M13 & M30 & M32 & M34 & E43 & E44 & E63 & E71 ;%{SE}%MKUKATPVW %CVW_SPS %VFBPSPS %P 2:FB PSPS = M13 & M30 & M32 & M34 & E43 & E44 & E63 & E71,3:FBPSPS
      ;ENDFOLD
      ;FOLD {H}
         VW_MPARA_ACT=P20_D
         Act_P1 = P20
         Act_P2 = P20
         VW(#MPARA,TRUE)
         SPS_FERTIG=FALSE
         TRIGGER WHEN DISTANCE=1 DELAY=0 DO SPS_TRIG(10021) PRIO=-1 UP_TIME_OUT=SPS_TIMEOUT
         LIN P20 C_DIS
         $ADVANCE=1
      ;ENDFOLD
   ;ENDFOLD
   ;FOLD KLIN VB=200[mm/s] Genau=40[mm] ACC=50% RobWzg=1 Base=2 SPSTrig=0[1/100s] P ;%{P}%MKUKATPVW,%CMOVE8,%VKLIN,%P 1:4, 2: VB=, 3:200, 4:[mm/s], 5: Genau=, 6:40, 7:[mm], 8: ACC=, 9:50, 10:%, 11: RobWzg=, 12:1, 13: Base=, 14:2, 15: SPSTrig=, 16:0, 17:[1/100s], 18: P, 19:21, 20:-1, 21:22
      ;FOLD 1: FB PSPS = M13 & M30 & M32 & M34 & E43 & E44 & E63 & E71 ;%{SE}%MKUKATPVW %CVW_SPS %VFBPSPS %P 2:FB PSPS = M13 & M30 & M32 & M34 & E43 & E44 & E63 & E71,3:FBPSPS
      ;ENDFOLD
      ;FOLD {H}
         VW_MPARA_ACT=P21_D
         Act_P1 = P21
         Act_P2 = P21
         VW(#MPARA,TRUE)
         SPS_FERTIG=FALSE
         TRIGGER WHEN DISTANCE=1 DELAY=0 DO SPS_TRIG(10022) PRIO=-1 UP_TIME_OUT=SPS_TIMEOUT
         LIN P21 C_DIS
         $ADVANCE=1
      ;ENDFOLD
   ;ENDFOLD
   ;FOLD -- Schaltpunkt 6 -- ;%{PSE}%MKUKATPVW,%CVW_COM,%VCOMMENT,%P 1:Comment:, 2:Schaltpunkt 6
      ;FOLD {H}
         M_COMMENT("Schaltpunkt 6")
      ;ENDFOLD
   ;ENDFOLD
   ;FOLD KLIN VB=200[mm/s] Genau=40[mm] ACC=50% RobWzg=1 Base=2 SPSTrig=0[1/100s] P ;%{P}%MKUKATPVW,%CMOVE8,%VKLIN,%P 1:4, 2: VB=, 3:200, 4:[mm/s], 5: Genau=, 6:40, 7:[mm], 8: ACC=, 9:50, 10:%, 11: RobWzg=, 12:1, 13: Base=, 14:2, 15: SPSTrig=, 16:0, 17:[1/100s], 18: P, 19:22, 20:-1, 21:23
      ;FOLD BS bin11 ( EIN ) = 6 Schaltpkt:5[mm]:-50[ms] ;%{SE}%MKUKATPVW %CVW_SPS %VBSARI %P 2:BS bin11 ( EIN ) = 6 Schaltpkt:5[mm]:-50[ms],3:BSARI
      ;ENDFOLD
      ;FOLD 1: FB PSPS = M13 & M30 & M32 & M34 & E43 & E44 & E63 & E71 ;%{SE}%MKUKATPVW %CVW_SPS %VFBPSPS %P 2:FB PSPS = M13 & M30 & M32 & M34 & E43 & E44 & E63 & E71,3:FBPSPS
      ;ENDFOLD
      ;FOLD {H}
         VW_MPARA_ACT=P22_D
         Act_P1 = P22
         Act_P2 = P22
         VW(#MPARA,TRUE)
         SPS_FERTIG=FALSE
         TRIGGER WHEN DISTANCE=1 DELAY=0 DO SPS_TRIG(10023) PRIO=-1 UP_TIME_OUT=SPS_TIMEOUT
         TRIGGER WHEN PATH=5 DELAY=-50 DO $B_OUT[11]=(6)
         LIN P22 C_DIS
         $ADVANCE=1
      ;ENDFOLD
   ;ENDFOLD
   ;FOLD KLIN VB=200[mm/s] Genau=40[mm] ACC=50% RobWzg=1 Base=2 SPSTrig=0[1/100s] P ;%{P}%MKUKATPVW,%CMOVE8,%VKLIN,%P 1:4, 2: VB=, 3:200, 4:[mm/s], 5: Genau=, 6:40, 7:[mm], 8: ACC=, 9:50, 10:%, 11: RobWzg=, 12:1, 13: Base=, 14:2, 15: SPSTrig=, 16:0, 17:[1/100s], 18: P, 19:23, 20:-1, 21:24
      ;FOLD 1: FB PSPS = M13 & M30 & M32 & M34 & E43 & E44 & E63 & E71 ;%{SE}%MKUKATPVW %CVW_SPS %VFBPSPS %P 2:FB PSPS = M13 & M30 & M32 & M34 & E43 & E44 & E63 & E71,3:FBPSPS
      ;ENDFOLD
      ;FOLD {H}
         VW_MPARA_ACT=P23_D
         Act_P1 = P23
         Act_P2 = P23
         VW(#MPARA,TRUE)
         SPS_FERTIG=FALSE
         TRIGGER WHEN DISTANCE=1 DELAY=0 DO SPS_TRIG(10024) PRIO=-1 UP_TIME_OUT=SPS_TIMEOUT
         LIN P23 C_DIS
         $ADVANCE=1
      ;ENDFOLD
   ;ENDFOLD
   ;FOLD KLIN VB=200[mm/s] Genau=40[mm] ACC=50% RobWzg=1 Base=2 SPSTrig=0[1/100s] P ;%{P}%MKUKATPVW,%CMOVE8,%VKLIN,%P 1:4, 2: VB=, 3:200, 4:[mm/s], 5: Genau=, 6:40, 7:[mm], 8: ACC=, 9:50, 10:%, 11: RobWzg=, 12:1, 13: Base=, 14:2, 15: SPSTrig=, 16:0, 17:[1/100s], 18: P, 19:24, 20:-1, 21:25
      ;FOLD 1: FB PSPS = M13 & M30 & M32 & M34 & E43 & E44 & E63 & E71 ;%{SE}%MKUKATPVW %CVW_SPS %VFBPSPS %P 2:FB PSPS = M13 & M30 & M32 & M34 & E43 & E44 & E63 & E71,3:FBPSPS
      ;ENDFOLD
      ;FOLD {H}
         VW_MPARA_ACT=P24_D
         Act_P1 = P24
         Act_P2 = P24
         VW(#MPARA,TRUE)
         SPS_FERTIG=FALSE
         TRIGGER WHEN DISTANCE=1 DELAY=0 DO SPS_TRIG(10025) PRIO=-1 UP_TIME_OUT=SPS_TIMEOUT
         LIN P24 C_DIS
         $ADVANCE=1
      ;ENDFOLD
   ;ENDFOLD
   ;FOLD KLIN VB=200[mm/s] Genau=40[mm] ACC=50% RobWzg=1 Base=2 SPSTrig=0[1/100s] P ;%{P}%MKUKATPVW,%CMOVE8,%VKLIN,%P 1:4, 2: VB=, 3:200, 4:[mm/s], 5: Genau=, 6:40, 7:[mm], 8: ACC=, 9:50, 10:%, 11: RobWzg=, 12:1, 13: Base=, 14:2, 15: SPSTrig=, 16:0, 17:[1/100s], 18: P, 19:25, 20:-1, 21:26
      ;FOLD 1: FB PSPS = M13 & M30 & M32 & M34 & E43 & E44 & E63 & E71 ;%{SE}%MKUKATPVW %CVW_SPS %VFBPSPS %P 2:FB PSPS = M13 & M30 & M32 & M34 & E43 & E44 & E63 & E71,3:FBPSPS
      ;ENDFOLD
      ;FOLD {H}
         VW_MPARA_ACT=P25_D
         Act_P1 = P25
         Act_P2 = P25
         VW(#MPARA,TRUE)
         SPS_FERTIG=FALSE
         TRIGGER WHEN DISTANCE=1 DELAY=0 DO SPS_TRIG(10026) PRIO=-1 UP_TIME_OUT=SPS_TIMEOUT
         LIN P25 C_DIS
         $ADVANCE=1
      ;ENDFOLD
   ;ENDFOLD
   ;FOLD KLIN VB=200[mm/s] Genau=40[mm] ACC=50% RobWzg=1 Base=2 SPSTrig=0[1/100s] P ;%{P}%MKUKATPVW,%CMOVE8,%VKLIN,%P 1:4, 2: VB=, 3:200, 4:[mm/s], 5: Genau=, 6:40, 7:[mm], 8: ACC=, 9:50, 10:%, 11: RobWzg=, 12:1, 13: Base=, 14:2, 15: SPSTrig=, 16:0, 17:[1/100s], 18: P, 19:26, 20:-1, 21:27
      ;FOLD 1: FB PSPS = M13 & M30 & M32 & M34 & E43 & E44 & E63 & E71 ;%{SE}%MKUKATPVW %CVW_SPS %VFBPSPS %P 2:FB PSPS = M13 & M30 & M32 & M34 & E43 & E44 & E63 & E71,3:FBPSPS
      ;ENDFOLD
      ;FOLD {H}
         VW_MPARA_ACT=P26_D
         Act_P1 = P26
         Act_P2 = P26
         VW(#MPARA,TRUE)
         SPS_FERTIG=FALSE
         TRIGGER WHEN DISTANCE=1 DELAY=0 DO SPS_TRIG(10027) PRIO=-1 UP_TIME_OUT=SPS_TIMEOUT
         LIN P26 C_DIS
         $ADVANCE=1
      ;ENDFOLD
   ;ENDFOLD
   ;FOLD KLIN VB=200[mm/s] Genau=40[mm] ACC=50% RobWzg=1 Base=2 SPSTrig=0[1/100s] P ;%{P}%MKUKATPVW,%CMOVE8,%VKLIN,%P 1:4, 2: VB=, 3:200, 4:[mm/s], 5: Genau=, 6:40, 7:[mm], 8: ACC=, 9:50, 10:%, 11: RobWzg=, 12:1, 13: Base=, 14:2, 15: SPSTrig=, 16:0, 17:[1/100s], 18: P, 19:27, 20:-1, 21:28
      ;FOLD 1: FB PSPS = M13 & M30 & M32 & M34 & E43 & E44 & E63 & E71 ;%{SE}%MKUKATPVW %CVW_SPS %VFBPSPS %P 2:FB PSPS = M13 & M30 & M32 & M34 & E43 & E44 & E63 & E71,3:FBPSPS
      ;ENDFOLD
      ;FOLD {H}
         VW_MPARA_ACT=P27_D
         Act_P1 = P27
         Act_P2 = P27
         VW(#MPARA,TRUE)
         SPS_FERTIG=FALSE
         TRIGGER WHEN DISTANCE=1 DELAY=0 DO SPS_TRIG(10028) PRIO=-1 UP_TIME_OUT=SPS_TIMEOUT
         LIN P27 C_DIS
         $ADVANCE=1
      ;ENDFOLD
   ;ENDFOLD
   ;FOLD KLIN VB=200[mm/s] Genau=40[mm] ACC=50% RobWzg=1 Base=2 SPSTrig=0[1/100s] P ;%{P}%MKUKATPVW,%CMOVE8,%VKLIN,%P 1:4, 2: VB=, 3:200, 4:[mm/s], 5: Genau=, 6:40, 7:[mm], 8: ACC=, 9:50, 10:%, 11: RobWzg=, 12:1, 13: Base=, 14:2, 15: SPSTrig=, 16:0, 17:[1/100s], 18: P, 19:28, 20:-1, 21:29
      ;FOLD 1: FB PSPS = M13 & M30 & M32 & M34 & E43 & E44 & E63 & E71 ;%{SE}%MKUKATPVW %CVW_SPS %VFBPSPS %P 2:FB PSPS = M13 & M30 & M32 & M34 & E43 & E44 & E63 & E71,3:FBPSPS
      ;ENDFOLD
      ;FOLD {H}
         VW_MPARA_ACT=P28_D
         Act_P1 = P28
         Act_P2 = P28
         VW(#MPARA,TRUE)
         SPS_FERTIG=FALSE
         TRIGGER WHEN DISTANCE=1 DELAY=0 DO SPS_TRIG(10029) PRIO=-1 UP_TIME_OUT=SPS_TIMEOUT
         LIN P28 C_DIS
         $ADVANCE=1
      ;ENDFOLD
   ;ENDFOLD
   ;FOLD -- Ende Klebenaht 5H4_833_055_C0002_A__1110_000100_LL -- ;%{PSE}%MKUKATPVW,%CVW_COM,%VCOMMENT,%P 1:Comment:, 2:Ende Klebenaht 5H4_833_055_C0002_A__1110_000100_LL
      ;FOLD {H}
         M_COMMENT("Ende Klebenaht 5H4_833_055_C0002_A__1110_000100_LL")
      ;ENDFOLD
   ;ENDFOLD
   ;FOLD -- Schaltpunkt 7 -- ;%{PSE}%MKUKATPVW,%CVW_COM,%VCOMMENT,%P 1:Comment:, 2:Schaltpunkt 7
      ;FOLD {H}
         M_COMMENT("Schaltpunkt 7")
      ;ENDFOLD
   ;ENDFOLD
   ;FOLD KLIN VB=200[mm/s] Genau=40[mm] ACC=50% RobWzg=1 Base=2 SPSTrig=5[1/100s] P ;%{P}%MKUKATPVW,%CMOVE8,%VKLIN,%P 1:4, 2: VB=, 3:200, 4:[mm/s], 5: Genau=, 6:40, 7:[mm], 8: ACC=, 9:50, 10:%, 11: RobWzg=, 12:1, 13: Base=, 14:2, 15: SPSTrig=, 16:5, 17:[1/100s], 18: P, 19:29, 20:-1, 21:30
      ;FOLD BS A1544 ( EIN ) = AUS Schaltpkt: 0 [mm]: -50 [ms] ;%{SE}%MKUKATPVW %CVW_SPS %VBSBO %P 2:BS A1544 ( EIN ) = AUS Schaltpkt: 0 [mm]: -50 [ms],3:BSBO
      ;ENDFOLD
      ;FOLD BS bin11 ( EIN ) = 7 Schaltpkt:5[mm]:-50[ms] ;%{SE}%MKUKATPVW %CVW_SPS %VBSARI %P 2:BS bin11 ( EIN ) = 7 Schaltpkt:5[mm]:-50[ms],3:BSARI
      ;ENDFOLD
      ;FOLD 1: FB PSPS = M13 & M30 & M32 & M34 & E43 & E44 & E63 & E71 ;%{SE}%MKUKATPVW %CVW_SPS %VFBPSPS %P 2:FB PSPS = M13 & M30 & M32 & M34 & E43 & E44 & E63 & E71,3:FBPSPS
      ;ENDFOLD
      ;FOLD {H}
         VW_MPARA_ACT=P29_D
         Act_P1 = P29
         Act_P2 = P29
         VW(#MPARA,TRUE)
         SPS_FERTIG=FALSE
         TRIGGER WHEN DISTANCE=1 DELAY=-50 DO SPS_TRIG(10030) PRIO=-1 UP_TIME_OUT=SPS_TIMEOUT
         TRIGGER WHEN PATH=0 DELAY=-50 DO $OUT[1544]=(FALSE)
         TRIGGER WHEN PATH=5 DELAY=-50 DO $B_OUT[11]=(7)
         LIN P29 C_DIS
         $ADVANCE=1
      ;ENDFOLD
   ;ENDFOLD
   ;FOLD KLIN VB=200[mm/s] Genau=40[mm] ACC=50% RobWzg=1 Base=2 SPSTrig=0[1/100s] P ;%{P}%MKUKATPVW,%CMOVE8,%VKLIN,%P 1:4, 2: VB=, 3:200, 4:[mm/s], 5: Genau=, 6:40, 7:[mm], 8: ACC=, 9:50, 10:%, 11: RobWzg=, 12:1, 13: Base=, 14:2, 15: SPSTrig=, 16:0, 17:[1/100s], 18: P, 19:30, 20:-1, 21:31
      ;FOLD 1: FB PSPS = M13 & M30 & M32 & M34 & E43 & E44 & E63 & E71 ;%{SE}%MKUKATPVW %CVW_SPS %VFBPSPS %P 2:FB PSPS = M13 & M30 & M32 & M34 & E43 & E44 & E63 & E71,3:FBPSPS
      ;ENDFOLD
      ;FOLD {H}
         VW_MPARA_ACT=P30_D
         Act_P1 = P30
         Act_P2 = P30
         VW(#MPARA,TRUE)
         SPS_FERTIG=FALSE
         TRIGGER WHEN DISTANCE=1 DELAY=0 DO SPS_TRIG(10031) PRIO=-1 UP_TIME_OUT=SPS_TIMEOUT
         LIN P30 C_DIS
         $ADVANCE=1
      ;ENDFOLD
   ;ENDFOLD
   ;FOLD KLIN VB=150[mm/s] Genau=30[mm] ACC=50% RobWzg=1 Base=2 SPSTrig=0[1/100s] P ;%{P}%MKUKATPVW,%CMOVE8,%VKLIN,%P 1:4, 2: VB=, 3:150, 4:[mm/s], 5: Genau=, 6:30, 7:[mm], 8: ACC=, 9:50, 10:%, 11: RobWzg=, 12:1, 13: Base=, 14:2, 15: SPSTrig=, 16:0, 17:[1/100s], 18: P, 19:31, 20:-1, 21:32
      ;FOLD 1: FB PSPS = M13 & M30 & M32 & M34 & E43 & E44 & E63 & E71 ;%{SE}%MKUKATPVW %CVW_SPS %VFBPSPS %P 2:FB PSPS = M13 & M30 & M32 & M34 & E43 & E44 & E63 & E71,3:FBPSPS
      ;ENDFOLD
      ;FOLD {H}
         VW_MPARA_ACT=P31_D
         Act_P1 = P31
         Act_P2 = P31
         VW(#MPARA,TRUE)
         SPS_FERTIG=FALSE
         TRIGGER WHEN DISTANCE=1 DELAY=0 DO SPS_TRIG(10032) PRIO=-1 UP_TIME_OUT=SPS_TIMEOUT
         LIN P31 C_DIS
         $ADVANCE=1
      ;ENDFOLD
   ;ENDFOLD
   ;FOLD -- Start Klebenaht 5H4_833_055_C0006_C__1150_000200_LL -- ;%{PSE}%MKUKATPVW,%CVW_COM,%VCOMMENT,%P 1:Comment:, 2:Start Klebenaht 5H4_833_055_C0006_C__1150_000200_LL
      ;FOLD {H}
         M_COMMENT("Start Klebenaht 5H4_833_055_C0006_C__1150_000200_LL")
      ;ENDFOLD
   ;ENDFOLD
   ;FOLD KLIN VB=150[mm/s] Genau=30[mm] ACC=50% RobWzg=1 Base=2 SPSTrig=5[1/100s] P ;%{P}%MKUKATPVW,%CMOVE8,%VKLIN,%P 1:4, 2: VB=, 3:150, 4:[mm/s], 5: Genau=, 6:30, 7:[mm], 8: ACC=, 9:50, 10:%, 11: RobWzg=, 12:1, 13: Base=, 14:2, 15: SPSTrig=, 16:5, 17:[1/100s], 18: P, 19:32, 20:-1, 21:33
      ;FOLD BS A1544 ( EIN ) = !E15 Schaltpkt:2[mm]:-50[ms] ;%{SE}%MKUKATPVW %CVW_SPS %VBSBO %P 2:BS A1544 ( EIN ) = !E15 Schaltpkt:2[mm]:-50[ms],3:BSBO
      ;ENDFOLD
      ;FOLD 1: FB PSPS = M13 & M30 & M32 & M34 & E43 & E44 & E63 & E71 ;%{SE}%MKUKATPVW %CVW_SPS %VFBPSPS %P 2:FB PSPS = M13 & M30 & M32 & M34 & E43 & E44 & E63 & E71,3:FBPSPS
      ;ENDFOLD
      ;FOLD {H}
         VW_MPARA_ACT=P32_D
         Act_P1 = P32
         Act_P2 = P32
         VW(#MPARA,TRUE)
         SPS_FERTIG=FALSE
         TRIGGER WHEN DISTANCE=1 DELAY=-50 DO SPS_TRIG(10033) PRIO=-1 UP_TIME_OUT=SPS_TIMEOUT
         TRIGGER WHEN PATH=2 DELAY=-50 DO $OUT[1544]=(NOT $IN[15])
         LIN P32 C_DIS
         $ADVANCE=1
      ;ENDFOLD
   ;ENDFOLD
   ;FOLD KLIN VB=150[mm/s] Genau=30[mm] ACC=50% RobWzg=1 Base=2 SPSTrig=0[1/100s] P ;%{P}%MKUKATPVW,%CMOVE8,%VKLIN,%P 1:4, 2: VB=, 3:150, 4:[mm/s], 5: Genau=, 6:30, 7:[mm], 8: ACC=, 9:50, 10:%, 11: RobWzg=, 12:1, 13: Base=, 14:2, 15: SPSTrig=, 16:0, 17:[1/100s], 18: P, 19:33, 20:-1, 21:34
      ;FOLD 1: FB PSPS = M13 & M30 & M32 & M34 & E43 & E44 & E63 & E71 ;%{SE}%MKUKATPVW %CVW_SPS %VFBPSPS %P 2:FB PSPS = M13 & M30 & M32 & M34 & E43 & E44 & E63 & E71,3:FBPSPS
      ;ENDFOLD
      ;FOLD {H}
         VW_MPARA_ACT=P33_D
         Act_P1 = P33
         Act_P2 = P33
         VW(#MPARA,TRUE)
         SPS_FERTIG=FALSE
         TRIGGER WHEN DISTANCE=1 DELAY=0 DO SPS_TRIG(10034) PRIO=-1 UP_TIME_OUT=SPS_TIMEOUT
         LIN P33 C_DIS
         $ADVANCE=1
      ;ENDFOLD
   ;ENDFOLD
   ;FOLD -- Ende Klebenaht 5H4_833_055_C0006_C__1150_000200_LL -- ;%{PSE}%MKUKATPVW,%CVW_COM,%VCOMMENT,%P 1:Comment:, 2:Ende Klebenaht 5H4_833_055_C0006_C__1150_000200_LL
      ;FOLD {H}
         M_COMMENT("Ende Klebenaht 5H4_833_055_C0006_C__1150_000200_LL")
      ;ENDFOLD
   ;ENDFOLD
   ;FOLD -- Schaltpunkt 8 -- ;%{PSE}%MKUKATPVW,%CVW_COM,%VCOMMENT,%P 1:Comment:, 2:Schaltpunkt 8
      ;FOLD {H}
         M_COMMENT("Schaltpunkt 8")
      ;ENDFOLD
   ;ENDFOLD
   ;FOLD KLIN VB=150[mm/s] Genau=30[mm] ACC=50% RobWzg=1 Base=2 SPSTrig=5[1/100s] P ;%{P}%MKUKATPVW,%CMOVE8,%VKLIN,%P 1:4, 2: VB=, 3:150, 4:[mm/s], 5: Genau=, 6:30, 7:[mm], 8: ACC=, 9:50, 10:%, 11: RobWzg=, 12:1, 13: Base=, 14:2, 15: SPSTrig=, 16:5, 17:[1/100s], 18: P, 19:34, 20:-1, 21:35
      ;FOLD BS A1544 ( EIN ) = AUS Schaltpkt:-1[mm]:-50[ms] ;%{SE}%MKUKATPVW %CVW_SPS %VBSBO %P 2:BS A1544 ( EIN ) = AUS Schaltpkt:-1[mm]:-50[ms],3:BSBO
      ;ENDFOLD
      ;FOLD BS bin11 ( EIN ) = 8 Schaltpkt:5[mm]:-50[ms] ;%{SE}%MKUKATPVW %CVW_SPS %VBSARI %P 2:BS bin11 ( EIN ) = 8 Schaltpkt:5[mm]:-50[ms],3:BSARI
      ;ENDFOLD
      ;FOLD 1: FB PSPS = M13 & M30 & M32 & M34 & E43 & E44 & E63 & E71 ;%{SE}%MKUKATPVW %CVW_SPS %VFBPSPS %P 2:FB PSPS = M13 & M30 & M32 & M34 & E43 & E44 & E63 & E71,3:FBPSPS
      ;ENDFOLD
      ;FOLD {H}
         VW_MPARA_ACT=P34_D
         Act_P1 = P34
         Act_P2 = P34
         VW(#MPARA,TRUE)
         SPS_FERTIG=FALSE
         TRIGGER WHEN DISTANCE=1 DELAY=-50 DO SPS_TRIG(10035) PRIO=-1 UP_TIME_OUT=SPS_TIMEOUT
         TRIGGER WHEN PATH=-1 DELAY=-50 DO $OUT[1544]=(FALSE)
         TRIGGER WHEN PATH=5 DELAY=-50 DO $B_OUT[11]=(8)
         LIN P34 C_DIS
         $ADVANCE=1
      ;ENDFOLD
   ;ENDFOLD
   ;FOLD KLIN VB=150[mm/s] Genau=30[mm] ACC=50% RobWzg=1 Base=2 SPSTrig=0[1/100s] P ;%{P}%MKUKATPVW,%CMOVE8,%VKLIN,%P 1:4, 2: VB=, 3:150, 4:[mm/s], 5: Genau=, 6:30, 7:[mm], 8: ACC=, 9:50, 10:%, 11: RobWzg=, 12:1, 13: Base=, 14:2, 15: SPSTrig=, 16:0, 17:[1/100s], 18: P, 19:35, 20:-1, 21:36
      ;FOLD 1: FB PSPS = M13 & M30 & M32 & M34 & E43 & E44 & E63 & E71 ;%{SE}%MKUKATPVW %CVW_SPS %VFBPSPS %P 2:FB PSPS = M13 & M30 & M32 & M34 & E43 & E44 & E63 & E71,3:FBPSPS
      ;ENDFOLD
      ;FOLD {H}
         VW_MPARA_ACT=P35_D
         Act_P1 = P35
         Act_P2 = P35
         VW(#MPARA,TRUE)
         SPS_FERTIG=FALSE
         TRIGGER WHEN DISTANCE=1 DELAY=0 DO SPS_TRIG(10036) PRIO=-1 UP_TIME_OUT=SPS_TIMEOUT
         LIN P35 C_DIS
         $ADVANCE=1
      ;ENDFOLD
   ;ENDFOLD
   ;FOLD LIN VB=300[mm/s] VE=10% ACC=50% RobWzg=1 Base=2 SPSTrig=0[1/100s] P ;%{P}%MKUKATPVW,%CMOVE8,%VLIN,%P 1:2, 2: VB=, 3:300, 4:[mm/s], 5: VE=, 6:10, 7:%, 8: ACC=, 9:50, 10:%, 11: RobWzg=, 12:1, 13: Base=, 14:2, 15: SPSTrig=, 16:0, 17:[1/100s], 18: P, 19:36, 20:-1, 21:37
      ;FOLD 1: FB PSPS = M13 & M30 & M32 & M34 & E43 & E44 & E63 & E71 ;%{SE}%MKUKATPVW %CVW_SPS %VFBPSPS %P 2:FB PSPS = M13 & M30 & M32 & M34 & E43 & E44 & E63 & E71,3:FBPSPS
      ;ENDFOLD
      ;FOLD {H}
         VW_MPARA_ACT=P36_D
         Act_P1 = P36
         Act_P2 = P36
         VW(#MPARA,TRUE)
         SPS_FERTIG=FALSE
         TRIGGER WHEN DISTANCE=1 DELAY=0 DO SPS_TRIG(10037) PRIO=-1 UP_TIME_OUT=SPS_TIMEOUT
         LIN P36 C_VEL
         $ADVANCE=1
      ;ENDFOLD
   ;ENDFOLD
   ;FOLD KLIN VB=200[mm/s] Genau=40[mm] ACC=50% RobWzg=1 Base=2 SPSTrig=0[1/100s] P ;%{P}%MKUKATPVW,%CMOVE8,%VKLIN,%P 1:4, 2: VB=, 3:200, 4:[mm/s], 5: Genau=, 6:40, 7:[mm], 8: ACC=, 9:50, 10:%, 11: RobWzg=, 12:1, 13: Base=, 14:2, 15: SPSTrig=, 16:0, 17:[1/100s], 18: P, 19:37, 20:-1, 21:38
      ;FOLD 1: FB PSPS = M13 & M30 & M32 & M34 & E43 & E44 & E63 & E71 ;%{SE}%MKUKATPVW %CVW_SPS %VFBPSPS %P 2:FB PSPS = M13 & M30 & M32 & M34 & E43 & E44 & E63 & E71,3:FBPSPS
      ;ENDFOLD
      ;FOLD {H}
         VW_MPARA_ACT=P37_D
         Act_P1 = P37
         Act_P2 = P37
         VW(#MPARA,TRUE)
         SPS_FERTIG=FALSE
         TRIGGER WHEN DISTANCE=1 DELAY=0 DO SPS_TRIG(10038) PRIO=-1 UP_TIME_OUT=SPS_TIMEOUT
         LIN P37 C_DIS
         $ADVANCE=1
      ;ENDFOLD
   ;ENDFOLD
   ;FOLD -- Start Klebenaht 5H4_833_055_C0005_D__1110_000400_LL -- ;%{PSE}%MKUKATPVW,%CVW_COM,%VCOMMENT,%P 1:Comment:, 2:Start Klebenaht 5H4_833_055_C0005_D__1110_000400_LL
      ;FOLD {H}
         M_COMMENT("Start Klebenaht 5H4_833_055_C0005_D__1110_000400_LL")
      ;ENDFOLD
   ;ENDFOLD
   ;FOLD KLIN VB=200[mm/s] Genau=40[mm] ACC=50% RobWzg=1 Base=2 SPSTrig=5[1/100s] P ;%{P}%MKUKATPVW,%CMOVE8,%VKLIN,%P 1:4, 2: VB=, 3:200, 4:[mm/s], 5: Genau=, 6:40, 7:[mm], 8: ACC=, 9:50, 10:%, 11: RobWzg=, 12:1, 13: Base=, 14:2, 15: SPSTrig=, 16:5, 17:[1/100s], 18: P, 19:38, 20:-1, 21:39
      ;FOLD BS A1544 ( EIN ) = !E15 Schaltpkt:2[mm]:-50[ms] ;%{SE}%MKUKATPVW %CVW_SPS %VBSBO %P 2:BS A1544 ( EIN ) = !E15 Schaltpkt:2[mm]:-50[ms],3:BSBO
      ;ENDFOLD
      ;FOLD 1: FB PSPS = M13 & M30 & M32 & M34 & E43 & E44 & E63 & E71 ;%{SE}%MKUKATPVW %CVW_SPS %VFBPSPS %P 2:FB PSPS = M13 & M30 & M32 & M34 & E43 & E44 & E63 & E71,3:FBPSPS
      ;ENDFOLD
      ;FOLD {H}
         VW_MPARA_ACT=P38_D
         Act_P1 = P38
         Act_P2 = P38
         VW(#MPARA,TRUE)
         SPS_FERTIG=FALSE
         TRIGGER WHEN DISTANCE=1 DELAY=-50 DO SPS_TRIG(10039) PRIO=-1 UP_TIME_OUT=SPS_TIMEOUT
         TRIGGER WHEN PATH=2 DELAY=-50 DO $OUT[1544]=(NOT $IN[15])
         LIN P38 C_DIS
         $ADVANCE=1
      ;ENDFOLD
   ;ENDFOLD
   ;FOLD KLIN VB=200[mm/s] Genau=40[mm] ACC=50% RobWzg=1 Base=2 SPSTrig=0[1/100s] P ;%{P}%MKUKATPVW,%CMOVE8,%VKLIN,%P 1:4, 2: VB=, 3:200, 4:[mm/s], 5: Genau=, 6:40, 7:[mm], 8: ACC=, 9:50, 10:%, 11: RobWzg=, 12:1, 13: Base=, 14:2, 15: SPSTrig=, 16:0, 17:[1/100s], 18: P, 19:39, 20:-1, 21:40
      ;FOLD 1: FB PSPS = M13 & M30 & M32 & M34 & E43 & E44 & E63 & E71 ;%{SE}%MKUKATPVW %CVW_SPS %VFBPSPS %P 2:FB PSPS = M13 & M30 & M32 & M34 & E43 & E44 & E63 & E71,3:FBPSPS
      ;ENDFOLD
      ;FOLD {H}
         VW_MPARA_ACT=P39_D
         Act_P1 = P39
         Act_P2 = P39
         VW(#MPARA,TRUE)
         SPS_FERTIG=FALSE
         TRIGGER WHEN DISTANCE=1 DELAY=0 DO SPS_TRIG(10040) PRIO=-1 UP_TIME_OUT=SPS_TIMEOUT
         LIN P39 C_DIS
         $ADVANCE=1
      ;ENDFOLD
   ;ENDFOLD
   ;FOLD KLIN VB=200[mm/s] Genau=40[mm] ACC=50% RobWzg=1 Base=2 SPSTrig=0[1/100s] P ;%{P}%MKUKATPVW,%CMOVE8,%VKLIN,%P 1:4, 2: VB=, 3:200, 4:[mm/s], 5: Genau=, 6:40, 7:[mm], 8: ACC=, 9:50, 10:%, 11: RobWzg=, 12:1, 13: Base=, 14:2, 15: SPSTrig=, 16:0, 17:[1/100s], 18: P, 19:40, 20:-1, 21:41
      ;FOLD 1: FB PSPS = M13 & M30 & M32 & M34 & E43 & E44 & E63 & E71 ;%{SE}%MKUKATPVW %CVW_SPS %VFBPSPS %P 2:FB PSPS = M13 & M30 & M32 & M34 & E43 & E44 & E63 & E71,3:FBPSPS
      ;ENDFOLD
      ;FOLD {H}
         VW_MPARA_ACT=P40_D
         Act_P1 = P40
         Act_P2 = P40
         VW(#MPARA,TRUE)
         SPS_FERTIG=FALSE
         TRIGGER WHEN DISTANCE=1 DELAY=0 DO SPS_TRIG(10041) PRIO=-1 UP_TIME_OUT=SPS_TIMEOUT
         LIN P40 C_DIS
         $ADVANCE=1
      ;ENDFOLD
   ;ENDFOLD
   ;FOLD KLIN VB=200[mm/s] Genau=40[mm] ACC=50% RobWzg=1 Base=2 SPSTrig=0[1/100s] P ;%{P}%MKUKATPVW,%CMOVE8,%VKLIN,%P 1:4, 2: VB=, 3:200, 4:[mm/s], 5: Genau=, 6:40, 7:[mm], 8: ACC=, 9:50, 10:%, 11: RobWzg=, 12:1, 13: Base=, 14:2, 15: SPSTrig=, 16:0, 17:[1/100s], 18: P, 19:41, 20:-1, 21:42
      ;FOLD 1: FB PSPS = M13 & M30 & M32 & M34 & E43 & E44 & E63 & E71 ;%{SE}%MKUKATPVW %CVW_SPS %VFBPSPS %P 2:FB PSPS = M13 & M30 & M32 & M34 & E43 & E44 & E63 & E71,3:FBPSPS
      ;ENDFOLD
      ;FOLD {H}
         VW_MPARA_ACT=P41_D
         Act_P1 = P41
         Act_P2 = P41
         VW(#MPARA,TRUE)
         SPS_FERTIG=FALSE
         TRIGGER WHEN DISTANCE=1 DELAY=0 DO SPS_TRIG(10042) PRIO=-1 UP_TIME_OUT=SPS_TIMEOUT
         LIN P41 C_DIS
         $ADVANCE=1
      ;ENDFOLD
   ;ENDFOLD
   ;FOLD KLIN VB=200[mm/s] Genau=40[mm] ACC=50% RobWzg=1 Base=2 SPSTrig=0[1/100s] P ;%{P}%MKUKATPVW,%CMOVE8,%VKLIN,%P 1:4, 2: VB=, 3:200, 4:[mm/s], 5: Genau=, 6:40, 7:[mm], 8: ACC=, 9:50, 10:%, 11: RobWzg=, 12:1, 13: Base=, 14:2, 15: SPSTrig=, 16:0, 17:[1/100s], 18: P, 19:42, 20:-1, 21:43
      ;FOLD 1: FB PSPS = M13 & M30 & M32 & M34 & E43 & E44 & E63 & E71 ;%{SE}%MKUKATPVW %CVW_SPS %VFBPSPS %P 2:FB PSPS = M13 & M30 & M32 & M34 & E43 & E44 & E63 & E71,3:FBPSPS
      ;ENDFOLD
      ;FOLD {H}
         VW_MPARA_ACT=P42_D
         Act_P1 = P42
         Act_P2 = P42
         VW(#MPARA,TRUE)
         SPS_FERTIG=FALSE
         TRIGGER WHEN DISTANCE=1 DELAY=0 DO SPS_TRIG(10043) PRIO=-1 UP_TIME_OUT=SPS_TIMEOUT
         LIN P42 C_DIS
         $ADVANCE=1
      ;ENDFOLD
   ;ENDFOLD
   ;FOLD KLIN VB=200[mm/s] Genau=40[mm] ACC=50% RobWzg=1 Base=2 SPSTrig=0[1/100s] P ;%{P}%MKUKATPVW,%CMOVE8,%VKLIN,%P 1:4, 2: VB=, 3:200, 4:[mm/s], 5: Genau=, 6:40, 7:[mm], 8: ACC=, 9:50, 10:%, 11: RobWzg=, 12:1, 13: Base=, 14:2, 15: SPSTrig=, 16:0, 17:[1/100s], 18: P, 19:43, 20:-1, 21:44
      ;FOLD 1: FB PSPS = M13 & M30 & M32 & M34 & E43 & E44 & E63 & E71 ;%{SE}%MKUKATPVW %CVW_SPS %VFBPSPS %P 2:FB PSPS = M13 & M30 & M32 & M34 & E43 & E44 & E63 & E71,3:FBPSPS
      ;ENDFOLD
      ;FOLD {H}
         VW_MPARA_ACT=P43_D
         Act_P1 = P43
         Act_P2 = P43
         VW(#MPARA,TRUE)
         SPS_FERTIG=FALSE
         TRIGGER WHEN DISTANCE=1 DELAY=0 DO SPS_TRIG(10044) PRIO=-1 UP_TIME_OUT=SPS_TIMEOUT
         LIN P43 C_DIS
         $ADVANCE=1
      ;ENDFOLD
   ;ENDFOLD
   ;FOLD KLIN VB=200[mm/s] Genau=40[mm] ACC=50% RobWzg=1 Base=2 SPSTrig=0[1/100s] P ;%{P}%MKUKATPVW,%CMOVE8,%VKLIN,%P 1:4, 2: VB=, 3:200, 4:[mm/s], 5: Genau=, 6:40, 7:[mm], 8: ACC=, 9:50, 10:%, 11: RobWzg=, 12:1, 13: Base=, 14:2, 15: SPSTrig=, 16:0, 17:[1/100s], 18: P, 19:44, 20:-1, 21:45
      ;FOLD 1: FB PSPS = M13 & M30 & M32 & M34 & E43 & E44 & E63 & E71 ;%{SE}%MKUKATPVW %CVW_SPS %VFBPSPS %P 2:FB PSPS = M13 & M30 & M32 & M34 & E43 & E44 & E63 & E71,3:FBPSPS
      ;ENDFOLD
      ;FOLD {H}
         VW_MPARA_ACT=P44_D
         Act_P1 = P44
         Act_P2 = P44
         VW(#MPARA,TRUE)
         SPS_FERTIG=FALSE
         TRIGGER WHEN DISTANCE=1 DELAY=0 DO SPS_TRIG(10045) PRIO=-1 UP_TIME_OUT=SPS_TIMEOUT
         LIN P44 C_DIS
         $ADVANCE=1
      ;ENDFOLD
   ;ENDFOLD
   ;FOLD -- Schaltpunkt 9 -- ;%{PSE}%MKUKATPVW,%CVW_COM,%VCOMMENT,%P 1:Comment:, 2:Schaltpunkt 9
      ;FOLD {H}
         M_COMMENT("Schaltpunkt 9")
      ;ENDFOLD
   ;ENDFOLD
   ;FOLD KLIN VB=200[mm/s] Genau=40[mm] ACC=50% RobWzg=1 Base=2 SPSTrig=0[1/100s] P ;%{P}%MKUKATPVW,%CMOVE8,%VKLIN,%P 1:4, 2: VB=, 3:200, 4:[mm/s], 5: Genau=, 6:40, 7:[mm], 8: ACC=, 9:50, 10:%, 11: RobWzg=, 12:1, 13: Base=, 14:2, 15: SPSTrig=, 16:0, 17:[1/100s], 18: P, 19:45, 20:-1, 21:46
      ;FOLD BS bin11 ( EIN ) = 9 Schaltpkt:5[mm]:-50[ms] ;%{SE}%MKUKATPVW %CVW_SPS %VBSARI %P 2:BS bin11 ( EIN ) = 9 Schaltpkt:5[mm]:-50[ms],3:BSARI
      ;ENDFOLD
      ;FOLD 1: FB PSPS = M13 & M30 & M32 & M34 & E43 & E44 & E63 & E71 ;%{SE}%MKUKATPVW %CVW_SPS %VFBPSPS %P 2:FB PSPS = M13 & M30 & M32 & M34 & E43 & E44 & E63 & E71,3:FBPSPS
      ;ENDFOLD
      ;FOLD {H}
         VW_MPARA_ACT=P45_D
         Act_P1 = P45
         Act_P2 = P45
         VW(#MPARA,TRUE)
         SPS_FERTIG=FALSE
         TRIGGER WHEN DISTANCE=1 DELAY=0 DO SPS_TRIG(10046) PRIO=-1 UP_TIME_OUT=SPS_TIMEOUT
         TRIGGER WHEN PATH=5 DELAY=-50 DO $B_OUT[11]=(9)
         LIN P45 C_DIS
         $ADVANCE=1
      ;ENDFOLD
   ;ENDFOLD
   ;FOLD KLIN VB=200[mm/s] Genau=40[mm] ACC=50% RobWzg=1 Base=2 SPSTrig=0[1/100s] P ;%{P}%MKUKATPVW,%CMOVE8,%VKLIN,%P 1:4, 2: VB=, 3:200, 4:[mm/s], 5: Genau=, 6:40, 7:[mm], 8: ACC=, 9:50, 10:%, 11: RobWzg=, 12:1, 13: Base=, 14:2, 15: SPSTrig=, 16:0, 17:[1/100s], 18: P, 19:46, 20:-1, 21:47
      ;FOLD 1: FB PSPS = M13 & M30 & M32 & M34 & E43 & E44 & E63 & E71 ;%{SE}%MKUKATPVW %CVW_SPS %VFBPSPS %P 2:FB PSPS = M13 & M30 & M32 & M34 & E43 & E44 & E63 & E71,3:FBPSPS
      ;ENDFOLD
      ;FOLD {H}
         VW_MPARA_ACT=P46_D
         Act_P1 = P46
         Act_P2 = P46
         VW(#MPARA,TRUE)
         SPS_FERTIG=FALSE
         TRIGGER WHEN DISTANCE=1 DELAY=0 DO SPS_TRIG(10047) PRIO=-1 UP_TIME_OUT=SPS_TIMEOUT
         LIN P46 C_DIS
         $ADVANCE=1
      ;ENDFOLD
   ;ENDFOLD
   ;FOLD KLIN VB=200[mm/s] Genau=40[mm] ACC=50% RobWzg=1 Base=2 SPSTrig=0[1/100s] P ;%{P}%MKUKATPVW,%CMOVE8,%VKLIN,%P 1:4, 2: VB=, 3:200, 4:[mm/s], 5: Genau=, 6:40, 7:[mm], 8: ACC=, 9:50, 10:%, 11: RobWzg=, 12:1, 13: Base=, 14:2, 15: SPSTrig=, 16:0, 17:[1/100s], 18: P, 19:47, 20:-1, 21:48
      ;FOLD 1: FB PSPS = M13 & M30 & M32 & M34 & E43 & E44 & E63 & E71 ;%{SE}%MKUKATPVW %CVW_SPS %VFBPSPS %P 2:FB PSPS = M13 & M30 & M32 & M34 & E43 & E44 & E63 & E71,3:FBPSPS
      ;ENDFOLD
      ;FOLD {H}
         VW_MPARA_ACT=P47_D
         Act_P1 = P47
         Act_P2 = P47
         VW(#MPARA,TRUE)
         SPS_FERTIG=FALSE
         TRIGGER WHEN DISTANCE=1 DELAY=0 DO SPS_TRIG(10048) PRIO=-1 UP_TIME_OUT=SPS_TIMEOUT
         LIN P47 C_DIS
         $ADVANCE=1
      ;ENDFOLD
   ;ENDFOLD
   ;FOLD KLIN VB=200[mm/s] Genau=40[mm] ACC=50% RobWzg=1 Base=2 SPSTrig=0[1/100s] P ;%{P}%MKUKATPVW,%CMOVE8,%VKLIN,%P 1:4, 2: VB=, 3:200, 4:[mm/s], 5: Genau=, 6:40, 7:[mm], 8: ACC=, 9:50, 10:%, 11: RobWzg=, 12:1, 13: Base=, 14:2, 15: SPSTrig=, 16:0, 17:[1/100s], 18: P, 19:48, 20:-1, 21:49
      ;FOLD 1: FB PSPS = M13 & M30 & M32 & M34 & E43 & E44 & E63 & E71 ;%{SE}%MKUKATPVW %CVW_SPS %VFBPSPS %P 2:FB PSPS = M13 & M30 & M32 & M34 & E43 & E44 & E63 & E71,3:FBPSPS
      ;ENDFOLD
      ;FOLD {H}
         VW_MPARA_ACT=P48_D
         Act_P1 = P48
         Act_P2 = P48
         VW(#MPARA,TRUE)
         SPS_FERTIG=FALSE
         TRIGGER WHEN DISTANCE=1 DELAY=0 DO SPS_TRIG(10049) PRIO=-1 UP_TIME_OUT=SPS_TIMEOUT
         LIN P48 C_DIS
         $ADVANCE=1
      ;ENDFOLD
   ;ENDFOLD
   ;FOLD KLIN VB=200[mm/s] Genau=40[mm] ACC=50% RobWzg=1 Base=2 SPSTrig=0[1/100s] P ;%{P}%MKUKATPVW,%CMOVE8,%VKLIN,%P 1:4, 2: VB=, 3:200, 4:[mm/s], 5: Genau=, 6:40, 7:[mm], 8: ACC=, 9:50, 10:%, 11: RobWzg=, 12:1, 13: Base=, 14:2, 15: SPSTrig=, 16:0, 17:[1/100s], 18: P, 19:49, 20:-1, 21:50
      ;FOLD 1: FB PSPS = M13 & M30 & M32 & M34 & E43 & E44 & E63 & E71 ;%{SE}%MKUKATPVW %CVW_SPS %VFBPSPS %P 2:FB PSPS = M13 & M30 & M32 & M34 & E43 & E44 & E63 & E71,3:FBPSPS
      ;ENDFOLD
      ;FOLD {H}
         VW_MPARA_ACT=P49_D
         Act_P1 = P49
         Act_P2 = P49
         VW(#MPARA,TRUE)
         SPS_FERTIG=FALSE
         TRIGGER WHEN DISTANCE=1 DELAY=0 DO SPS_TRIG(10050) PRIO=-1 UP_TIME_OUT=SPS_TIMEOUT
         LIN P49 C_DIS
         $ADVANCE=1
      ;ENDFOLD
   ;ENDFOLD
   ;FOLD KLIN VB=200[mm/s] Genau=40[mm] ACC=50% RobWzg=1 Base=2 SPSTrig=0[1/100s] P ;%{P}%MKUKATPVW,%CMOVE8,%VKLIN,%P 1:4, 2: VB=, 3:200, 4:[mm/s], 5: Genau=, 6:40, 7:[mm], 8: ACC=, 9:50, 10:%, 11: RobWzg=, 12:1, 13: Base=, 14:2, 15: SPSTrig=, 16:0, 17:[1/100s], 18: P, 19:50, 20:-1, 21:51
      ;FOLD 1: FB PSPS = M13 & M30 & M32 & M34 & E43 & E44 & E63 & E71 ;%{SE}%MKUKATPVW %CVW_SPS %VFBPSPS %P 2:FB PSPS = M13 & M30 & M32 & M34 & E43 & E44 & E63 & E71,3:FBPSPS
      ;ENDFOLD
      ;FOLD {H}
         VW_MPARA_ACT=P50_D
         Act_P1 = P50
         Act_P2 = P50
         VW(#MPARA,TRUE)
         SPS_FERTIG=FALSE
         TRIGGER WHEN DISTANCE=1 DELAY=0 DO SPS_TRIG(10051) PRIO=-1 UP_TIME_OUT=SPS_TIMEOUT
         LIN P50 C_DIS
         $ADVANCE=1
      ;ENDFOLD
   ;ENDFOLD
   ;FOLD KLIN VB=200[mm/s] Genau=40[mm] ACC=50% RobWzg=1 Base=2 SPSTrig=0[1/100s] P ;%{P}%MKUKATPVW,%CMOVE8,%VKLIN,%P 1:4, 2: VB=, 3:200, 4:[mm/s], 5: Genau=, 6:40, 7:[mm], 8: ACC=, 9:50, 10:%, 11: RobWzg=, 12:1, 13: Base=, 14:2, 15: SPSTrig=, 16:0, 17:[1/100s], 18: P, 19:51, 20:-1, 21:52
      ;FOLD 1: FB PSPS = M13 & M30 & M32 & M34 & E43 & E44 & E63 & E71 ;%{SE}%MKUKATPVW %CVW_SPS %VFBPSPS %P 2:FB PSPS = M13 & M30 & M32 & M34 & E43 & E44 & E63 & E71,3:FBPSPS
      ;ENDFOLD
      ;FOLD {H}
         VW_MPARA_ACT=P51_D
         Act_P1 = P51
         Act_P2 = P51
         VW(#MPARA,TRUE)
         SPS_FERTIG=FALSE
         TRIGGER WHEN DISTANCE=1 DELAY=0 DO SPS_TRIG(10052) PRIO=-1 UP_TIME_OUT=SPS_TIMEOUT
         LIN P51 C_DIS
         $ADVANCE=1
      ;ENDFOLD
   ;ENDFOLD
   ;FOLD KLIN VB=200[mm/s] Genau=40[mm] ACC=50% RobWzg=1 Base=2 SPSTrig=0[1/100s] P ;%{P}%MKUKATPVW,%CMOVE8,%VKLIN,%P 1:4, 2: VB=, 3:200, 4:[mm/s], 5: Genau=, 6:40, 7:[mm], 8: ACC=, 9:50, 10:%, 11: RobWzg=, 12:1, 13: Base=, 14:2, 15: SPSTrig=, 16:0, 17:[1/100s], 18: P, 19:52, 20:-1, 21:53
      ;FOLD 1: FB PSPS = M13 & M30 & M32 & M34 & E43 & E44 & E63 & E71 ;%{SE}%MKUKATPVW %CVW_SPS %VFBPSPS %P 2:FB PSPS = M13 & M30 & M32 & M34 & E43 & E44 & E63 & E71,3:FBPSPS
      ;ENDFOLD
      ;FOLD {H}
         VW_MPARA_ACT=P52_D
         Act_P1 = P52
         Act_P2 = P52
         VW(#MPARA,TRUE)
         SPS_FERTIG=FALSE
         TRIGGER WHEN DISTANCE=1 DELAY=0 DO SPS_TRIG(10053) PRIO=-1 UP_TIME_OUT=SPS_TIMEOUT
         LIN P52 C_DIS
         $ADVANCE=1
      ;ENDFOLD
   ;ENDFOLD
   ;FOLD KLIN VB=200[mm/s] Genau=40[mm] ACC=50% RobWzg=1 Base=2 SPSTrig=0[1/100s] P ;%{P}%MKUKATPVW,%CMOVE8,%VKLIN,%P 1:4, 2: VB=, 3:200, 4:[mm/s], 5: Genau=, 6:40, 7:[mm], 8: ACC=, 9:50, 10:%, 11: RobWzg=, 12:1, 13: Base=, 14:2, 15: SPSTrig=, 16:0, 17:[1/100s], 18: P, 19:53, 20:-1, 21:54
      ;FOLD 1: FB PSPS = M13 & M30 & M32 & M34 & E43 & E44 & E63 & E71 ;%{SE}%MKUKATPVW %CVW_SPS %VFBPSPS %P 2:FB PSPS = M13 & M30 & M32 & M34 & E43 & E44 & E63 & E71,3:FBPSPS
      ;ENDFOLD
      ;FOLD {H}
         VW_MPARA_ACT=P53_D
         Act_P1 = P53
         Act_P2 = P53
         VW(#MPARA,TRUE)
         SPS_FERTIG=FALSE
         TRIGGER WHEN DISTANCE=1 DELAY=0 DO SPS_TRIG(10054) PRIO=-1 UP_TIME_OUT=SPS_TIMEOUT
         LIN P53 C_DIS
         $ADVANCE=1
      ;ENDFOLD
   ;ENDFOLD
   ;FOLD -- Schaltpunkt 10 -- ;%{PSE}%MKUKATPVW,%CVW_COM,%VCOMMENT,%P 1:Comment:, 2:Schaltpunkt 10
      ;FOLD {H}
         M_COMMENT("Schaltpunkt 10")
      ;ENDFOLD
   ;ENDFOLD
   ;FOLD KLIN VB=200[mm/s] Genau=40[mm] ACC=50% RobWzg=1 Base=2 SPSTrig=0[1/100s] P ;%{P}%MKUKATPVW,%CMOVE8,%VKLIN,%P 1:4, 2: VB=, 3:200, 4:[mm/s], 5: Genau=, 6:40, 7:[mm], 8: ACC=, 9:50, 10:%, 11: RobWzg=, 12:1, 13: Base=, 14:2, 15: SPSTrig=, 16:0, 17:[1/100s], 18: P, 19:54, 20:-1, 21:55
      ;FOLD BS bin11 ( EIN ) = 10 Schaltpkt:5[mm]:-50[ms] ;%{SE}%MKUKATPVW %CVW_SPS %VBSARI %P 2:BS bin11 ( EIN ) = 10 Schaltpkt:5[mm]:-50[ms],3:BSARI
      ;ENDFOLD
      ;FOLD 1: FB PSPS = M13 & M30 & M32 & M34 & E43 & E44 & E63 & E71 ;%{SE}%MKUKATPVW %CVW_SPS %VFBPSPS %P 2:FB PSPS = M13 & M30 & M32 & M34 & E43 & E44 & E63 & E71,3:FBPSPS
      ;ENDFOLD
      ;FOLD {H}
         VW_MPARA_ACT=P54_D
         Act_P1 = P54
         Act_P2 = P54
         VW(#MPARA,TRUE)
         SPS_FERTIG=FALSE
         TRIGGER WHEN DISTANCE=1 DELAY=0 DO SPS_TRIG(10055) PRIO=-1 UP_TIME_OUT=SPS_TIMEOUT
         TRIGGER WHEN PATH=5 DELAY=-50 DO $B_OUT[11]=(10)
         LIN P54 C_DIS
         $ADVANCE=1
      ;ENDFOLD
   ;ENDFOLD
   ;FOLD KLIN VB=200[mm/s] Genau=40[mm] ACC=50% RobWzg=1 Base=2 SPSTrig=0[1/100s] P ;%{P}%MKUKATPVW,%CMOVE8,%VKLIN,%P 1:4, 2: VB=, 3:200, 4:[mm/s], 5: Genau=, 6:40, 7:[mm], 8: ACC=, 9:50, 10:%, 11: RobWzg=, 12:1, 13: Base=, 14:2, 15: SPSTrig=, 16:0, 17:[1/100s], 18: P, 19:55, 20:-1, 21:56
      ;FOLD 1: FB PSPS = M13 & M30 & M32 & M34 & E43 & E44 & E63 & E71 ;%{SE}%MKUKATPVW %CVW_SPS %VFBPSPS %P 2:FB PSPS = M13 & M30 & M32 & M34 & E43 & E44 & E63 & E71,3:FBPSPS
      ;ENDFOLD
      ;FOLD {H}
         VW_MPARA_ACT=P55_D
         Act_P1 = P55
         Act_P2 = P55
         VW(#MPARA,TRUE)
         SPS_FERTIG=FALSE
         TRIGGER WHEN DISTANCE=1 DELAY=0 DO SPS_TRIG(10056) PRIO=-1 UP_TIME_OUT=SPS_TIMEOUT
         LIN P55 C_DIS
         $ADVANCE=1
      ;ENDFOLD
   ;ENDFOLD
   ;FOLD KLIN VB=200[mm/s] Genau=40[mm] ACC=50% RobWzg=1 Base=2 SPSTrig=0[1/100s] P ;%{P}%MKUKATPVW,%CMOVE8,%VKLIN,%P 1:4, 2: VB=, 3:200, 4:[mm/s], 5: Genau=, 6:40, 7:[mm], 8: ACC=, 9:50, 10:%, 11: RobWzg=, 12:1, 13: Base=, 14:2, 15: SPSTrig=, 16:0, 17:[1/100s], 18: P, 19:56, 20:-1, 21:57
      ;FOLD 1: FB PSPS = M13 & M30 & M32 & M34 & E43 & E44 & E63 & E71 ;%{SE}%MKUKATPVW %CVW_SPS %VFBPSPS %P 2:FB PSPS = M13 & M30 & M32 & M34 & E43 & E44 & E63 & E71,3:FBPSPS
      ;ENDFOLD
      ;FOLD {H}
         VW_MPARA_ACT=P56_D
         Act_P1 = P56
         Act_P2 = P56
         VW(#MPARA,TRUE)
         SPS_FERTIG=FALSE
         TRIGGER WHEN DISTANCE=1 DELAY=0 DO SPS_TRIG(10057) PRIO=-1 UP_TIME_OUT=SPS_TIMEOUT
         LIN P56 C_DIS
         $ADVANCE=1
      ;ENDFOLD
   ;ENDFOLD
   ;FOLD KLIN VB=200[mm/s] Genau=40[mm] ACC=50% RobWzg=1 Base=2 SPSTrig=0[1/100s] P ;%{P}%MKUKATPVW,%CMOVE8,%VKLIN,%P 1:4, 2: VB=, 3:200, 4:[mm/s], 5: Genau=, 6:40, 7:[mm], 8: ACC=, 9:50, 10:%, 11: RobWzg=, 12:1, 13: Base=, 14:2, 15: SPSTrig=, 16:0, 17:[1/100s], 18: P, 19:57, 20:-1, 21:58
      ;FOLD 1: FB PSPS = M13 & M30 & M32 & M34 & E43 & E44 & E63 & E71 ;%{SE}%MKUKATPVW %CVW_SPS %VFBPSPS %P 2:FB PSPS = M13 & M30 & M32 & M34 & E43 & E44 & E63 & E71,3:FBPSPS
      ;ENDFOLD
      ;FOLD {H}
         VW_MPARA_ACT=P57_D
         Act_P1 = P57
         Act_P2 = P57
         VW(#MPARA,TRUE)
         SPS_FERTIG=FALSE
         TRIGGER WHEN DISTANCE=1 DELAY=0 DO SPS_TRIG(10058) PRIO=-1 UP_TIME_OUT=SPS_TIMEOUT
         LIN P57 C_DIS
         $ADVANCE=1
      ;ENDFOLD
   ;ENDFOLD
   ;FOLD KLIN VB=200[mm/s] Genau=40[mm] ACC=50% RobWzg=1 Base=2 SPSTrig=0[1/100s] P ;%{P}%MKUKATPVW,%CMOVE8,%VKLIN,%P 1:4, 2: VB=, 3:200, 4:[mm/s], 5: Genau=, 6:40, 7:[mm], 8: ACC=, 9:50, 10:%, 11: RobWzg=, 12:1, 13: Base=, 14:2, 15: SPSTrig=, 16:0, 17:[1/100s], 18: P, 19:58, 20:-1, 21:59
      ;FOLD 1: FB PSPS = M13 & M30 & M32 & M34 & E43 & E44 & E63 & E71 ;%{SE}%MKUKATPVW %CVW_SPS %VFBPSPS %P 2:FB PSPS = M13 & M30 & M32 & M34 & E43 & E44 & E63 & E71,3:FBPSPS
      ;ENDFOLD
      ;FOLD {H}
         VW_MPARA_ACT=P58_D
         Act_P1 = P58
         Act_P2 = P58
         VW(#MPARA,TRUE)
         SPS_FERTIG=FALSE
         TRIGGER WHEN DISTANCE=1 DELAY=0 DO SPS_TRIG(10059) PRIO=-1 UP_TIME_OUT=SPS_TIMEOUT
         LIN P58 C_DIS
         $ADVANCE=1
      ;ENDFOLD
   ;ENDFOLD
   ;FOLD KLIN VB=200[mm/s] Genau=40[mm] ACC=50% RobWzg=1 Base=2 SPSTrig=0[1/100s] P ;%{P}%MKUKATPVW,%CMOVE8,%VKLIN,%P 1:4, 2: VB=, 3:200, 4:[mm/s], 5: Genau=, 6:40, 7:[mm], 8: ACC=, 9:50, 10:%, 11: RobWzg=, 12:1, 13: Base=, 14:2, 15: SPSTrig=, 16:0, 17:[1/100s], 18: P, 19:59, 20:-1, 21:60
      ;FOLD 1: FB PSPS = M13 & M30 & M32 & M34 & E43 & E44 & E63 & E71 ;%{SE}%MKUKATPVW %CVW_SPS %VFBPSPS %P 2:FB PSPS = M13 & M30 & M32 & M34 & E43 & E44 & E63 & E71,3:FBPSPS
      ;ENDFOLD
      ;FOLD {H}
         VW_MPARA_ACT=P59_D
         Act_P1 = P59
         Act_P2 = P59
         VW(#MPARA,TRUE)
         SPS_FERTIG=FALSE
         TRIGGER WHEN DISTANCE=1 DELAY=0 DO SPS_TRIG(10060) PRIO=-1 UP_TIME_OUT=SPS_TIMEOUT
         LIN P59 C_DIS
         $ADVANCE=1
      ;ENDFOLD
   ;ENDFOLD
   ;FOLD KLIN VB=200[mm/s] Genau=40[mm] ACC=50% RobWzg=1 Base=2 SPSTrig=0[1/100s] P ;%{P}%MKUKATPVW,%CMOVE8,%VKLIN,%P 1:4, 2: VB=, 3:200, 4:[mm/s], 5: Genau=, 6:40, 7:[mm], 8: ACC=, 9:50, 10:%, 11: RobWzg=, 12:1, 13: Base=, 14:2, 15: SPSTrig=, 16:0, 17:[1/100s], 18: P, 19:60, 20:-1, 21:61
      ;FOLD 1: FB PSPS = M13 & M30 & M32 & M34 & E43 & E44 & E63 & E71 ;%{SE}%MKUKATPVW %CVW_SPS %VFBPSPS %P 2:FB PSPS = M13 & M30 & M32 & M34 & E43 & E44 & E63 & E71,3:FBPSPS
      ;ENDFOLD
      ;FOLD {H}
         VW_MPARA_ACT=P60_D
         Act_P1 = P60
         Act_P2 = P60
         VW(#MPARA,TRUE)
         SPS_FERTIG=FALSE
         TRIGGER WHEN DISTANCE=1 DELAY=0 DO SPS_TRIG(10061) PRIO=-1 UP_TIME_OUT=SPS_TIMEOUT
         LIN P60 C_DIS
         $ADVANCE=1
      ;ENDFOLD
   ;ENDFOLD
   ;FOLD KLIN VB=200[mm/s] Genau=40[mm] ACC=50% RobWzg=1 Base=2 SPSTrig=0[1/100s] P ;%{P}%MKUKATPVW,%CMOVE8,%VKLIN,%P 1:4, 2: VB=, 3:200, 4:[mm/s], 5: Genau=, 6:40, 7:[mm], 8: ACC=, 9:50, 10:%, 11: RobWzg=, 12:1, 13: Base=, 14:2, 15: SPSTrig=, 16:0, 17:[1/100s], 18: P, 19:61, 20:-1, 21:62
      ;FOLD 1: FB PSPS = M13 & M30 & M32 & M34 & E43 & E44 & E63 & E71 ;%{SE}%MKUKATPVW %CVW_SPS %VFBPSPS %P 2:FB PSPS = M13 & M30 & M32 & M34 & E43 & E44 & E63 & E71,3:FBPSPS
      ;ENDFOLD
      ;FOLD {H}
         VW_MPARA_ACT=P61_D
         Act_P1 = P61
         Act_P2 = P61
         VW(#MPARA,TRUE)
         SPS_FERTIG=FALSE
         TRIGGER WHEN DISTANCE=1 DELAY=0 DO SPS_TRIG(10062) PRIO=-1 UP_TIME_OUT=SPS_TIMEOUT
         LIN P61 C_DIS
         $ADVANCE=1
      ;ENDFOLD
   ;ENDFOLD
   ;FOLD KLIN VB=200[mm/s] Genau=40[mm] ACC=50% RobWzg=1 Base=2 SPSTrig=0[1/100s] P ;%{P}%MKUKATPVW,%CMOVE8,%VKLIN,%P 1:4, 2: VB=, 3:200, 4:[mm/s], 5: Genau=, 6:40, 7:[mm], 8: ACC=, 9:50, 10:%, 11: RobWzg=, 12:1, 13: Base=, 14:2, 15: SPSTrig=, 16:0, 17:[1/100s], 18: P, 19:62, 20:-1, 21:63
      ;FOLD 1: FB PSPS = M13 & M30 & M32 & M34 & E43 & E44 & E63 & E71 ;%{SE}%MKUKATPVW %CVW_SPS %VFBPSPS %P 2:FB PSPS = M13 & M30 & M32 & M34 & E43 & E44 & E63 & E71,3:FBPSPS
      ;ENDFOLD
      ;FOLD {H}
         VW_MPARA_ACT=P62_D
         Act_P1 = P62
         Act_P2 = P62
         VW(#MPARA,TRUE)
         SPS_FERTIG=FALSE
         TRIGGER WHEN DISTANCE=1 DELAY=0 DO SPS_TRIG(10063) PRIO=-1 UP_TIME_OUT=SPS_TIMEOUT
         LIN P62 C_DIS
         $ADVANCE=1
      ;ENDFOLD
   ;ENDFOLD
   ;FOLD KLIN VB=200[mm/s] Genau=40[mm] ACC=50% RobWzg=1 Base=2 SPSTrig=0[1/100s] P ;%{P}%MKUKATPVW,%CMOVE8,%VKLIN,%P 1:4, 2: VB=, 3:200, 4:[mm/s], 5: Genau=, 6:40, 7:[mm], 8: ACC=, 9:50, 10:%, 11: RobWzg=, 12:1, 13: Base=, 14:2, 15: SPSTrig=, 16:0, 17:[1/100s], 18: P, 19:63, 20:-1, 21:64
      ;FOLD 1: FB PSPS = M13 & M30 & M32 & M34 & E43 & E44 & E63 & E71 ;%{SE}%MKUKATPVW %CVW_SPS %VFBPSPS %P 2:FB PSPS = M13 & M30 & M32 & M34 & E43 & E44 & E63 & E71,3:FBPSPS
      ;ENDFOLD
      ;FOLD {H}
         VW_MPARA_ACT=P63_D
         Act_P1 = P63
         Act_P2 = P63
         VW(#MPARA,TRUE)
         SPS_FERTIG=FALSE
         TRIGGER WHEN DISTANCE=1 DELAY=0 DO SPS_TRIG(10064) PRIO=-1 UP_TIME_OUT=SPS_TIMEOUT
         LIN P63 C_DIS
         $ADVANCE=1
      ;ENDFOLD
   ;ENDFOLD
   ;FOLD KLIN VB=200[mm/s] Genau=40[mm] ACC=50% RobWzg=1 Base=2 SPSTrig=0[1/100s] P ;%{P}%MKUKATPVW,%CMOVE8,%VKLIN,%P 1:4, 2: VB=, 3:200, 4:[mm/s], 5: Genau=, 6:40, 7:[mm], 8: ACC=, 9:50, 10:%, 11: RobWzg=, 12:1, 13: Base=, 14:2, 15: SPSTrig=, 16:0, 17:[1/100s], 18: P, 19:64, 20:-1, 21:65
      ;FOLD 1: FB PSPS = M13 & M30 & M32 & M34 & E43 & E44 & E63 & E71 ;%{SE}%MKUKATPVW %CVW_SPS %VFBPSPS %P 2:FB PSPS = M13 & M30 & M32 & M34 & E43 & E44 & E63 & E71,3:FBPSPS
      ;ENDFOLD
      ;FOLD {H}
         VW_MPARA_ACT=P64_D
         Act_P1 = P64
         Act_P2 = P64
         VW(#MPARA,TRUE)
         SPS_FERTIG=FALSE
         TRIGGER WHEN DISTANCE=1 DELAY=0 DO SPS_TRIG(10065) PRIO=-1 UP_TIME_OUT=SPS_TIMEOUT
         LIN P64 C_DIS
         $ADVANCE=1
      ;ENDFOLD
   ;ENDFOLD
   ;FOLD -- Schaltpunkt 11 -- ;%{PSE}%MKUKATPVW,%CVW_COM,%VCOMMENT,%P 1:Comment:, 2:Schaltpunkt 11
      ;FOLD {H}
         M_COMMENT("Schaltpunkt 11")
      ;ENDFOLD
   ;ENDFOLD
   ;FOLD KLIN VB=200[mm/s] Genau=40[mm] ACC=50% RobWzg=1 Base=2 SPSTrig=0[1/100s] P ;%{P}%MKUKATPVW,%CMOVE8,%VKLIN,%P 1:4, 2: VB=, 3:200, 4:[mm/s], 5: Genau=, 6:40, 7:[mm], 8: ACC=, 9:50, 10:%, 11: RobWzg=, 12:1, 13: Base=, 14:2, 15: SPSTrig=, 16:0, 17:[1/100s], 18: P, 19:65, 20:-1, 21:66
      ;FOLD BS bin11 ( EIN ) = 11 Schaltpkt:5[mm]:-50[ms] ;%{SE}%MKUKATPVW %CVW_SPS %VBSARI %P 2:BS bin11 ( EIN ) = 11 Schaltpkt:5[mm]:-50[ms],3:BSARI
      ;ENDFOLD
      ;FOLD 1: FB PSPS = M13 & M30 & M32 & M34 & E43 & E44 & E63 & E71 ;%{SE}%MKUKATPVW %CVW_SPS %VFBPSPS %P 2:FB PSPS = M13 & M30 & M32 & M34 & E43 & E44 & E63 & E71,3:FBPSPS
      ;ENDFOLD
      ;FOLD {H}
         VW_MPARA_ACT=P65_D
         Act_P1 = P65
         Act_P2 = P65
         VW(#MPARA,TRUE)
         SPS_FERTIG=FALSE
         TRIGGER WHEN DISTANCE=1 DELAY=0 DO SPS_TRIG(10066) PRIO=-1 UP_TIME_OUT=SPS_TIMEOUT
         TRIGGER WHEN PATH=5 DELAY=-50 DO $B_OUT[11]=(11)
         LIN P65 C_DIS
         $ADVANCE=1
      ;ENDFOLD
   ;ENDFOLD
   ;FOLD KLIN VB=200[mm/s] Genau=40[mm] ACC=50% RobWzg=1 Base=2 SPSTrig=0[1/100s] P ;%{P}%MKUKATPVW,%CMOVE8,%VKLIN,%P 1:4, 2: VB=, 3:200, 4:[mm/s], 5: Genau=, 6:40, 7:[mm], 8: ACC=, 9:50, 10:%, 11: RobWzg=, 12:1, 13: Base=, 14:2, 15: SPSTrig=, 16:0, 17:[1/100s], 18: P, 19:66, 20:-1, 21:67
      ;FOLD 1: FB PSPS = M13 & M30 & M32 & M34 & E43 & E44 & E63 & E71 ;%{SE}%MKUKATPVW %CVW_SPS %VFBPSPS %P 2:FB PSPS = M13 & M30 & M32 & M34 & E43 & E44 & E63 & E71,3:FBPSPS
      ;ENDFOLD
      ;FOLD {H}
         VW_MPARA_ACT=P66_D
         Act_P1 = P66
         Act_P2 = P66
         VW(#MPARA,TRUE)
         SPS_FERTIG=FALSE
         TRIGGER WHEN DISTANCE=1 DELAY=0 DO SPS_TRIG(10067) PRIO=-1 UP_TIME_OUT=SPS_TIMEOUT
         LIN P66 C_DIS
         $ADVANCE=1
      ;ENDFOLD
   ;ENDFOLD
   ;FOLD KLIN VB=200[mm/s] Genau=40[mm] ACC=50% RobWzg=1 Base=2 SPSTrig=0[1/100s] P ;%{P}%MKUKATPVW,%CMOVE8,%VKLIN,%P 1:4, 2: VB=, 3:200, 4:[mm/s], 5: Genau=, 6:40, 7:[mm], 8: ACC=, 9:50, 10:%, 11: RobWzg=, 12:1, 13: Base=, 14:2, 15: SPSTrig=, 16:0, 17:[1/100s], 18: P, 19:67, 20:-1, 21:68
      ;FOLD 1: FB PSPS = M13 & M30 & M32 & M34 & E43 & E44 & E63 & E71 ;%{SE}%MKUKATPVW %CVW_SPS %VFBPSPS %P 2:FB PSPS = M13 & M30 & M32 & M34 & E43 & E44 & E63 & E71,3:FBPSPS
      ;ENDFOLD
      ;FOLD {H}
         VW_MPARA_ACT=P67_D
         Act_P1 = P67
         Act_P2 = P67
         VW(#MPARA,TRUE)
         SPS_FERTIG=FALSE
         TRIGGER WHEN DISTANCE=1 DELAY=0 DO SPS_TRIG(10068) PRIO=-1 UP_TIME_OUT=SPS_TIMEOUT
         LIN P67 C_DIS
         $ADVANCE=1
      ;ENDFOLD
   ;ENDFOLD
   ;FOLD KLIN VB=200[mm/s] Genau=40[mm] ACC=50% RobWzg=1 Base=2 SPSTrig=0[1/100s] P ;%{P}%MKUKATPVW,%CMOVE8,%VKLIN,%P 1:4, 2: VB=, 3:200, 4:[mm/s], 5: Genau=, 6:40, 7:[mm], 8: ACC=, 9:50, 10:%, 11: RobWzg=, 12:1, 13: Base=, 14:2, 15: SPSTrig=, 16:0, 17:[1/100s], 18: P, 19:68, 20:-1, 21:69
      ;FOLD 1: FB PSPS = M13 & M30 & M32 & M34 & E43 & E44 & E63 & E71 ;%{SE}%MKUKATPVW %CVW_SPS %VFBPSPS %P 2:FB PSPS = M13 & M30 & M32 & M34 & E43 & E44 & E63 & E71,3:FBPSPS
      ;ENDFOLD
      ;FOLD {H}
         VW_MPARA_ACT=P68_D
         Act_P1 = P68
         Act_P2 = P68
         VW(#MPARA,TRUE)
         SPS_FERTIG=FALSE
         TRIGGER WHEN DISTANCE=1 DELAY=0 DO SPS_TRIG(10069) PRIO=-1 UP_TIME_OUT=SPS_TIMEOUT
         LIN P68 C_DIS
         $ADVANCE=1
      ;ENDFOLD
   ;ENDFOLD
   ;FOLD KLIN VB=200[mm/s] Genau=40[mm] ACC=50% RobWzg=1 Base=2 SPSTrig=0[1/100s] P ;%{P}%MKUKATPVW,%CMOVE8,%VKLIN,%P 1:4, 2: VB=, 3:200, 4:[mm/s], 5: Genau=, 6:40, 7:[mm], 8: ACC=, 9:50, 10:%, 11: RobWzg=, 12:1, 13: Base=, 14:2, 15: SPSTrig=, 16:0, 17:[1/100s], 18: P, 19:69, 20:-1, 21:70
      ;FOLD 1: FB PSPS = M13 & M30 & M32 & M34 & E43 & E44 & E63 & E71 ;%{SE}%MKUKATPVW %CVW_SPS %VFBPSPS %P 2:FB PSPS = M13 & M30 & M32 & M34 & E43 & E44 & E63 & E71,3:FBPSPS
      ;ENDFOLD
      ;FOLD {H}
         VW_MPARA_ACT=P69_D
         Act_P1 = P69
         Act_P2 = P69
         VW(#MPARA,TRUE)
         SPS_FERTIG=FALSE
         TRIGGER WHEN DISTANCE=1 DELAY=0 DO SPS_TRIG(10070) PRIO=-1 UP_TIME_OUT=SPS_TIMEOUT
         LIN P69 C_DIS
         $ADVANCE=1
      ;ENDFOLD
   ;ENDFOLD
   ;FOLD KLIN VB=200[mm/s] Genau=40[mm] ACC=50% RobWzg=1 Base=2 SPSTrig=0[1/100s] P ;%{P}%MKUKATPVW,%CMOVE8,%VKLIN,%P 1:4, 2: VB=, 3:200, 4:[mm/s], 5: Genau=, 6:40, 7:[mm], 8: ACC=, 9:50, 10:%, 11: RobWzg=, 12:1, 13: Base=, 14:2, 15: SPSTrig=, 16:0, 17:[1/100s], 18: P, 19:70, 20:-1, 21:71
      ;FOLD 1: FB PSPS = M13 & M30 & M32 & M34 & E43 & E44 & E63 & E71 ;%{SE}%MKUKATPVW %CVW_SPS %VFBPSPS %P 2:FB PSPS = M13 & M30 & M32 & M34 & E43 & E44 & E63 & E71,3:FBPSPS
      ;ENDFOLD
      ;FOLD {H}
         VW_MPARA_ACT=P70_D
         Act_P1 = P70
         Act_P2 = P70
         VW(#MPARA,TRUE)
         SPS_FERTIG=FALSE
         TRIGGER WHEN DISTANCE=1 DELAY=0 DO SPS_TRIG(10071) PRIO=-1 UP_TIME_OUT=SPS_TIMEOUT
         LIN P70 C_DIS
         $ADVANCE=1
      ;ENDFOLD
   ;ENDFOLD
   ;FOLD KLIN VB=200[mm/s] Genau=40[mm] ACC=50% RobWzg=1 Base=2 SPSTrig=0[1/100s] P ;%{P}%MKUKATPVW,%CMOVE8,%VKLIN,%P 1:4, 2: VB=, 3:200, 4:[mm/s], 5: Genau=, 6:40, 7:[mm], 8: ACC=, 9:50, 10:%, 11: RobWzg=, 12:1, 13: Base=, 14:2, 15: SPSTrig=, 16:0, 17:[1/100s], 18: P, 19:71, 20:-1, 21:72
      ;FOLD 1: FB PSPS = M13 & M30 & M32 & M34 & E43 & E44 & E63 & E71 ;%{SE}%MKUKATPVW %CVW_SPS %VFBPSPS %P 2:FB PSPS = M13 & M30 & M32 & M34 & E43 & E44 & E63 & E71,3:FBPSPS
      ;ENDFOLD
      ;FOLD {H}
         VW_MPARA_ACT=P71_D
         Act_P1 = P71
         Act_P2 = P71
         VW(#MPARA,TRUE)
         SPS_FERTIG=FALSE
         TRIGGER WHEN DISTANCE=1 DELAY=0 DO SPS_TRIG(10072) PRIO=-1 UP_TIME_OUT=SPS_TIMEOUT
         LIN P71 C_DIS
         $ADVANCE=1
      ;ENDFOLD
   ;ENDFOLD
   ;FOLD -- Ende Klebenaht 5H4_833_055_C0005_D__1110_000400_LL -- ;%{PSE}%MKUKATPVW,%CVW_COM,%VCOMMENT,%P 1:Comment:, 2:Ende Klebenaht 5H4_833_055_C0005_D__1110_000400_LL
      ;FOLD {H}
         M_COMMENT("Ende Klebenaht 5H4_833_055_C0005_D__1110_000400_LL")
      ;ENDFOLD
   ;ENDFOLD
   ;FOLD -- Schaltpunkt 12 -- ;%{PSE}%MKUKATPVW,%CVW_COM,%VCOMMENT,%P 1:Comment:, 2:Schaltpunkt 12
      ;FOLD {H}
         M_COMMENT("Schaltpunkt 12")
      ;ENDFOLD
   ;ENDFOLD
   ;FOLD KLIN VB=200[mm/s] Genau=40[mm] ACC=50% RobWzg=1 Base=2 SPSTrig=5[1/100s] P ;%{P}%MKUKATPVW,%CMOVE8,%VKLIN,%P 1:4, 2: VB=, 3:200, 4:[mm/s], 5: Genau=, 6:40, 7:[mm], 8: ACC=, 9:50, 10:%, 11: RobWzg=, 12:1, 13: Base=, 14:2, 15: SPSTrig=, 16:5, 17:[1/100s], 18: P, 19:72, 20:-1, 21:73
      ;FOLD BS A1544 ( EIN ) = AUS Schaltpkt:-1[mm]:-50[ms] ;%{SE}%MKUKATPVW %CVW_SPS %VBSBO %P 2:BS A1544 ( EIN ) = AUS Schaltpkt:-1[mm]:-50[ms],3:BSBO
      ;ENDFOLD
      ;FOLD BS bin11 ( EIN ) = 12 Schaltpkt:5[mm]:-50[ms] ;%{SE}%MKUKATPVW %CVW_SPS %VBSARI %P 2:BS bin11 ( EIN ) = 12 Schaltpkt:5[mm]:-50[ms],3:BSARI
      ;ENDFOLD
      ;FOLD 1: FB PSPS = M13 & M30 & M32 & M34 & E43 & E44 & E63 & E71 ;%{SE}%MKUKATPVW %CVW_SPS %VFBPSPS %P 2:FB PSPS = M13 & M30 & M32 & M34 & E43 & E44 & E63 & E71,3:FBPSPS
      ;ENDFOLD
      ;FOLD {H}
         VW_MPARA_ACT=P72_D
         Act_P1 = P72
         Act_P2 = P72
         VW(#MPARA,TRUE)
         SPS_FERTIG=FALSE
         TRIGGER WHEN DISTANCE=1 DELAY=-50 DO SPS_TRIG(10073) PRIO=-1 UP_TIME_OUT=SPS_TIMEOUT
         TRIGGER WHEN PATH=-1 DELAY=-50 DO $OUT[1544]=(FALSE)
         TRIGGER WHEN PATH=5 DELAY=-50 DO $B_OUT[11]=(12)
         LIN P72 C_DIS
         $ADVANCE=1
      ;ENDFOLD
   ;ENDFOLD
   ;FOLD KLIN VB=200[mm/s] Genau=40[mm] ACC=50% RobWzg=1 Base=2 SPSTrig=0[1/100s] P ;%{P}%MKUKATPVW,%CMOVE8,%VKLIN,%P 1:4, 2: VB=, 3:200, 4:[mm/s], 5: Genau=, 6:40, 7:[mm], 8: ACC=, 9:50, 10:%, 11: RobWzg=, 12:1, 13: Base=, 14:2, 15: SPSTrig=, 16:0, 17:[1/100s], 18: P, 19:73, 20:-1, 21:74
      ;FOLD 1: FB PSPS = M13 & M30 & M32 & M34 & E43 & E44 & E63 & E71 ;%{SE}%MKUKATPVW %CVW_SPS %VFBPSPS %P 2:FB PSPS = M13 & M30 & M32 & M34 & E43 & E44 & E63 & E71,3:FBPSPS
      ;ENDFOLD
      ;FOLD {H}
         VW_MPARA_ACT=P73_D
         Act_P1 = P73
         Act_P2 = P73
         VW(#MPARA,TRUE)
         SPS_FERTIG=FALSE
         TRIGGER WHEN DISTANCE=1 DELAY=0 DO SPS_TRIG(10074) PRIO=-1 UP_TIME_OUT=SPS_TIMEOUT
         LIN P73 C_DIS
         $ADVANCE=1
      ;ENDFOLD
   ;ENDFOLD
   ;FOLD PTP VB=100% VE=100% ACC=100% RobWzg=1 Base=2 SPSTrig=0[1/100s] P ;%{P}%MKUKATPVW,%CMOVE8,%VPTP,%P 1:1, 2: VB=, 3:100, 4:%, 5: VE=, 6:100, 7:%, 8: ACC=, 9:100, 10:%, 11: RobWzg=, 12:1, 13: Base=, 14:2, 15: SPSTrig=, 16:0, 17:[1/100s], 18: P, 19:74, 20:-1, 21:75
      ;FOLD 1: FB PSPS = M13 & M30 & M32 & M34 & E43 & E44 & E63 & E71 ;%{SE}%MKUKATPVW %CVW_SPS %VFBPSPS %P 2:FB PSPS = M13 & M30 & M32 & M34 & E43 & E44 & E63 & E71,3:FBPSPS
      ;ENDFOLD
      ;FOLD {H}
         VW_MPARA_ACT=P74_D
         Act_P1 = P74
         Act_P2 = P74
         VW(#MPARA,TRUE)
         SPS_FERTIG=FALSE
         TRIGGER WHEN DISTANCE=1 DELAY=0 DO SPS_TRIG(10075) PRIO=-1 UP_TIME_OUT=SPS_TIMEOUT
         PTP P74 C_PTP C_VEL
         $ADVANCE=1
      ;ENDFOLD
   ;ENDFOLD
   ;FOLD PTP VB=100% VE=100% ACC=100% RobWzg=1 Base=2 SPSTrig=0[1/100s] P ;%{P}%MKUKATPVW,%CMOVE8,%VPTP,%P 1:1, 2: VB=, 3:100, 4:%, 5: VE=, 6:100, 7:%, 8: ACC=, 9:100, 10:%, 11: RobWzg=, 12:1, 13: Base=, 14:2, 15: SPSTrig=, 16:0, 17:[1/100s], 18: P, 19:75, 20:-1, 21:76
      ;FOLD 1: FB PSPS = M13 & M30 & M32 & M34 & E43 & E44 & E63 & E71 ;%{SE}%MKUKATPVW %CVW_SPS %VFBPSPS %P 2:FB PSPS = M13 & M30 & M32 & M34 & E43 & E44 & E63 & E71,3:FBPSPS
      ;ENDFOLD
      ;FOLD {H}
         VW_MPARA_ACT=P75_D
         Act_P1 = P75
         Act_P2 = P75
         VW(#MPARA,TRUE)
         SPS_FERTIG=FALSE
         TRIGGER WHEN DISTANCE=1 DELAY=0 DO SPS_TRIG(10076) PRIO=-1 UP_TIME_OUT=SPS_TIMEOUT
         PTP P75 C_PTP C_VEL
         $ADVANCE=1
      ;ENDFOLD
   ;ENDFOLD
   ;FOLD KLIN VB=200[mm/s] Genau=40[mm] ACC=50% RobWzg=1 Base=2 SPSTrig=0[1/100s] P ;%{P}%MKUKATPVW,%CMOVE8,%VKLIN,%P 1:4, 2: VB=, 3:200, 4:[mm/s], 5: Genau=, 6:40, 7:[mm], 8: ACC=, 9:50, 10:%, 11: RobWzg=, 12:1, 13: Base=, 14:2, 15: SPSTrig=, 16:0, 17:[1/100s], 18: P, 19:76, 20:-1, 21:77
      ;FOLD 1: FB PSPS = M13 & M30 & M32 & M34 & E43 & E44 & E63 & E71 ;%{SE}%MKUKATPVW %CVW_SPS %VFBPSPS %P 2:FB PSPS = M13 & M30 & M32 & M34 & E43 & E44 & E63 & E71,3:FBPSPS
      ;ENDFOLD
      ;FOLD {H}
         VW_MPARA_ACT=P76_D
         Act_P1 = P76
         Act_P2 = P76
         VW(#MPARA,TRUE)
         SPS_FERTIG=FALSE
         TRIGGER WHEN DISTANCE=1 DELAY=0 DO SPS_TRIG(10077) PRIO=-1 UP_TIME_OUT=SPS_TIMEOUT
         LIN P76 C_DIS
         $ADVANCE=1
      ;ENDFOLD
   ;ENDFOLD
   ;FOLD -- Start Klebenaht 5H4_833_055_C0005_D__1110_000500_LL -- ;%{PSE}%MKUKATPVW,%CVW_COM,%VCOMMENT,%P 1:Comment:, 2:Start Klebenaht 5H4_833_055_C0005_D__1110_000500_LL
      ;FOLD {H}
         M_COMMENT("Start Klebenaht 5H4_833_055_C0005_D__1110_000500_LL")
      ;ENDFOLD
   ;ENDFOLD
   ;FOLD KLIN VB=200[mm/s] Genau=40[mm] ACC=50% RobWzg=1 Base=2 SPSTrig=5[1/100s] P ;%{P}%MKUKATPVW,%CMOVE8,%VKLIN,%P 1:4, 2: VB=, 3:200, 4:[mm/s], 5: Genau=, 6:40, 7:[mm], 8: ACC=, 9:50, 10:%, 11: RobWzg=, 12:1, 13: Base=, 14:2, 15: SPSTrig=, 16:5, 17:[1/100s], 18: P, 19:77, 20:-1, 21:78
      ;FOLD BS A1544 ( EIN ) = !E15 Schaltpkt:2[mm]:-50[ms] ;%{SE}%MKUKATPVW %CVW_SPS %VBSBO %P 2:BS A1544 ( EIN ) = !E15 Schaltpkt:2[mm]:-50[ms],3:BSBO
      ;ENDFOLD
      ;FOLD 1: FB PSPS = M13 & M30 & M32 & M34 & E43 & E44 & E63 & E71 ;%{SE}%MKUKATPVW %CVW_SPS %VFBPSPS %P 2:FB PSPS = M13 & M30 & M32 & M34 & E43 & E44 & E63 & E71,3:FBPSPS
      ;ENDFOLD
      ;FOLD {H}
         VW_MPARA_ACT=P77_D
         Act_P1 = P77
         Act_P2 = P77
         VW(#MPARA,TRUE)
         SPS_FERTIG=FALSE
         TRIGGER WHEN DISTANCE=1 DELAY=-50 DO SPS_TRIG(10078) PRIO=-1 UP_TIME_OUT=SPS_TIMEOUT
         TRIGGER WHEN PATH=2 DELAY=-50 DO $OUT[1544]=(NOT $IN[15])
         LIN P77 C_DIS
         $ADVANCE=1
      ;ENDFOLD
   ;ENDFOLD
   ;FOLD KLIN VB=200[mm/s] Genau=40[mm] ACC=50% RobWzg=1 Base=2 SPSTrig=0[1/100s] P ;%{P}%MKUKATPVW,%CMOVE8,%VKLIN,%P 1:4, 2: VB=, 3:200, 4:[mm/s], 5: Genau=, 6:40, 7:[mm], 8: ACC=, 9:50, 10:%, 11: RobWzg=, 12:1, 13: Base=, 14:2, 15: SPSTrig=, 16:0, 17:[1/100s], 18: P, 19:78, 20:-1, 21:79
      ;FOLD 1: FB PSPS = M13 & M30 & M32 & M34 & E43 & E44 & E63 & E71 ;%{SE}%MKUKATPVW %CVW_SPS %VFBPSPS %P 2:FB PSPS = M13 & M30 & M32 & M34 & E43 & E44 & E63 & E71,3:FBPSPS
      ;ENDFOLD
      ;FOLD {H}
         VW_MPARA_ACT=P78_D
         Act_P1 = P78
         Act_P2 = P78
         VW(#MPARA,TRUE)
         SPS_FERTIG=FALSE
         TRIGGER WHEN DISTANCE=1 DELAY=0 DO SPS_TRIG(10079) PRIO=-1 UP_TIME_OUT=SPS_TIMEOUT
         LIN P78 C_DIS
         $ADVANCE=1
      ;ENDFOLD
   ;ENDFOLD
   ;FOLD KLIN VB=200[mm/s] Genau=40[mm] ACC=50% RobWzg=1 Base=2 SPSTrig=0[1/100s] P ;%{P}%MKUKATPVW,%CMOVE8,%VKLIN,%P 1:4, 2: VB=, 3:200, 4:[mm/s], 5: Genau=, 6:40, 7:[mm], 8: ACC=, 9:50, 10:%, 11: RobWzg=, 12:1, 13: Base=, 14:2, 15: SPSTrig=, 16:0, 17:[1/100s], 18: P, 19:79, 20:-1, 21:80
      ;FOLD 1: FB PSPS = M13 & M30 & M32 & M34 & E43 & E44 & E63 & E71 ;%{SE}%MKUKATPVW %CVW_SPS %VFBPSPS %P 2:FB PSPS = M13 & M30 & M32 & M34 & E43 & E44 & E63 & E71,3:FBPSPS
      ;ENDFOLD
      ;FOLD {H}
         VW_MPARA_ACT=P79_D
         Act_P1 = P79
         Act_P2 = P79
         VW(#MPARA,TRUE)
         SPS_FERTIG=FALSE
         TRIGGER WHEN DISTANCE=1 DELAY=0 DO SPS_TRIG(10080) PRIO=-1 UP_TIME_OUT=SPS_TIMEOUT
         LIN P79 C_DIS
         $ADVANCE=1
      ;ENDFOLD
   ;ENDFOLD
   ;FOLD KLIN VB=200[mm/s] Genau=40[mm] ACC=50% RobWzg=1 Base=2 SPSTrig=0[1/100s] P ;%{P}%MKUKATPVW,%CMOVE8,%VKLIN,%P 1:4, 2: VB=, 3:200, 4:[mm/s], 5: Genau=, 6:40, 7:[mm], 8: ACC=, 9:50, 10:%, 11: RobWzg=, 12:1, 13: Base=, 14:2, 15: SPSTrig=, 16:0, 17:[1/100s], 18: P, 19:80, 20:-1, 21:81
      ;FOLD 1: FB PSPS = M13 & M30 & M32 & M34 & E43 & E44 & E63 & E71 ;%{SE}%MKUKATPVW %CVW_SPS %VFBPSPS %P 2:FB PSPS = M13 & M30 & M32 & M34 & E43 & E44 & E63 & E71,3:FBPSPS
      ;ENDFOLD
      ;FOLD {H}
         VW_MPARA_ACT=P80_D
         Act_P1 = P80
         Act_P2 = P80
         VW(#MPARA,TRUE)
         SPS_FERTIG=FALSE
         TRIGGER WHEN DISTANCE=1 DELAY=0 DO SPS_TRIG(10081) PRIO=-1 UP_TIME_OUT=SPS_TIMEOUT
         LIN P80 C_DIS
         $ADVANCE=1
      ;ENDFOLD
   ;ENDFOLD
   ;FOLD -- Schaltpunkt 13 -- ;%{PSE}%MKUKATPVW,%CVW_COM,%VCOMMENT,%P 1:Comment:, 2:Schaltpunkt 13
      ;FOLD {H}
         M_COMMENT("Schaltpunkt 13")
      ;ENDFOLD
   ;ENDFOLD
   ;FOLD KLIN VB=200[mm/s] Genau=40[mm] ACC=50% RobWzg=1 Base=2 SPSTrig=0[1/100s] P ;%{P}%MKUKATPVW,%CMOVE8,%VKLIN,%P 1:4, 2: VB=, 3:200, 4:[mm/s], 5: Genau=, 6:40, 7:[mm], 8: ACC=, 9:50, 10:%, 11: RobWzg=, 12:1, 13: Base=, 14:2, 15: SPSTrig=, 16:0, 17:[1/100s], 18: P, 19:81, 20:-1, 21:82
      ;FOLD BS bin11 ( EIN ) = 13 Schaltpkt:5[mm]:-50[ms] ;%{SE}%MKUKATPVW %CVW_SPS %VBSARI %P 2:BS bin11 ( EIN ) = 13 Schaltpkt:5[mm]:-50[ms],3:BSARI
      ;ENDFOLD
      ;FOLD 1: FB PSPS = M13 & M30 & M32 & M34 & E43 & E44 & E63 & E71 ;%{SE}%MKUKATPVW %CVW_SPS %VFBPSPS %P 2:FB PSPS = M13 & M30 & M32 & M34 & E43 & E44 & E63 & E71,3:FBPSPS
      ;ENDFOLD
      ;FOLD {H}
         VW_MPARA_ACT=P81_D
         Act_P1 = P81
         Act_P2 = P81
         VW(#MPARA,TRUE)
         SPS_FERTIG=FALSE
         TRIGGER WHEN DISTANCE=1 DELAY=0 DO SPS_TRIG(10082) PRIO=-1 UP_TIME_OUT=SPS_TIMEOUT
         TRIGGER WHEN PATH=5 DELAY=-50 DO $B_OUT[11]=(13)
         LIN P81 C_DIS
         $ADVANCE=1
      ;ENDFOLD
   ;ENDFOLD
   ;FOLD KLIN VB=200[mm/s] Genau=40[mm] ACC=50% RobWzg=1 Base=2 SPSTrig=0[1/100s] P ;%{P}%MKUKATPVW,%CMOVE8,%VKLIN,%P 1:4, 2: VB=, 3:200, 4:[mm/s], 5: Genau=, 6:40, 7:[mm], 8: ACC=, 9:50, 10:%, 11: RobWzg=, 12:1, 13: Base=, 14:2, 15: SPSTrig=, 16:0, 17:[1/100s], 18: P, 19:82, 20:-1, 21:83
      ;FOLD 1: FB PSPS = M13 & M30 & M32 & M34 & E43 & E44 & E63 & E71 ;%{SE}%MKUKATPVW %CVW_SPS %VFBPSPS %P 2:FB PSPS = M13 & M30 & M32 & M34 & E43 & E44 & E63 & E71,3:FBPSPS
      ;ENDFOLD
      ;FOLD {H}
         VW_MPARA_ACT=P82_D
         Act_P1 = P82
         Act_P2 = P82
         VW(#MPARA,TRUE)
         SPS_FERTIG=FALSE
         TRIGGER WHEN DISTANCE=1 DELAY=0 DO SPS_TRIG(10083) PRIO=-1 UP_TIME_OUT=SPS_TIMEOUT
         LIN P82 C_DIS
         $ADVANCE=1
      ;ENDFOLD
   ;ENDFOLD
   ;FOLD KLIN VB=200[mm/s] Genau=40[mm] ACC=50% RobWzg=1 Base=2 SPSTrig=0[1/100s] P ;%{P}%MKUKATPVW,%CMOVE8,%VKLIN,%P 1:4, 2: VB=, 3:200, 4:[mm/s], 5: Genau=, 6:40, 7:[mm], 8: ACC=, 9:50, 10:%, 11: RobWzg=, 12:1, 13: Base=, 14:2, 15: SPSTrig=, 16:0, 17:[1/100s], 18: P, 19:83, 20:-1, 21:84
      ;FOLD 1: FB PSPS = M13 & M30 & M32 & M34 & E43 & E44 & E63 & E71 ;%{SE}%MKUKATPVW %CVW_SPS %VFBPSPS %P 2:FB PSPS = M13 & M30 & M32 & M34 & E43 & E44 & E63 & E71,3:FBPSPS
      ;ENDFOLD
      ;FOLD {H}
         VW_MPARA_ACT=P83_D
         Act_P1 = P83
         Act_P2 = P83
         VW(#MPARA,TRUE)
         SPS_FERTIG=FALSE
         TRIGGER WHEN DISTANCE=1 DELAY=0 DO SPS_TRIG(10084) PRIO=-1 UP_TIME_OUT=SPS_TIMEOUT
         LIN P83 C_DIS
         $ADVANCE=1
      ;ENDFOLD
   ;ENDFOLD
   ;FOLD KLIN VB=200[mm/s] Genau=40[mm] ACC=50% RobWzg=1 Base=2 SPSTrig=0[1/100s] P ;%{P}%MKUKATPVW,%CMOVE8,%VKLIN,%P 1:4, 2: VB=, 3:200, 4:[mm/s], 5: Genau=, 6:40, 7:[mm], 8: ACC=, 9:50, 10:%, 11: RobWzg=, 12:1, 13: Base=, 14:2, 15: SPSTrig=, 16:0, 17:[1/100s], 18: P, 19:84, 20:-1, 21:85
      ;FOLD 1: FB PSPS = M13 & M30 & M32 & M34 & E43 & E44 & E63 & E71 ;%{SE}%MKUKATPVW %CVW_SPS %VFBPSPS %P 2:FB PSPS = M13 & M30 & M32 & M34 & E43 & E44 & E63 & E71,3:FBPSPS
      ;ENDFOLD
      ;FOLD {H}
         VW_MPARA_ACT=P84_D
         Act_P1 = P84
         Act_P2 = P84
         VW(#MPARA,TRUE)
         SPS_FERTIG=FALSE
         TRIGGER WHEN DISTANCE=1 DELAY=0 DO SPS_TRIG(10085) PRIO=-1 UP_TIME_OUT=SPS_TIMEOUT
         LIN P84 C_DIS
         $ADVANCE=1
      ;ENDFOLD
   ;ENDFOLD
   ;FOLD -- Schaltpunkt 14 -- ;%{PSE}%MKUKATPVW,%CVW_COM,%VCOMMENT,%P 1:Comment:, 2:Schaltpunkt 14
      ;FOLD {H}
         M_COMMENT("Schaltpunkt 14")
      ;ENDFOLD
   ;ENDFOLD
   ;FOLD KLIN VB=200[mm/s] Genau=40[mm] ACC=50% RobWzg=1 Base=2 SPSTrig=0[1/100s] P ;%{P}%MKUKATPVW,%CMOVE8,%VKLIN,%P 1:4, 2: VB=, 3:200, 4:[mm/s], 5: Genau=, 6:40, 7:[mm], 8: ACC=, 9:50, 10:%, 11: RobWzg=, 12:1, 13: Base=, 14:2, 15: SPSTrig=, 16:0, 17:[1/100s], 18: P, 19:85, 20:-1, 21:86
      ;FOLD BS bin11 ( EIN ) = 14 Schaltpkt:5[mm]:-50[ms] ;%{SE}%MKUKATPVW %CVW_SPS %VBSARI %P 2:BS bin11 ( EIN ) = 14 Schaltpkt:5[mm]:-50[ms],3:BSARI
      ;ENDFOLD
      ;FOLD 1: FB PSPS = M13 & M30 & M32 & M34 & E43 & E44 & E63 & E71 ;%{SE}%MKUKATPVW %CVW_SPS %VFBPSPS %P 2:FB PSPS = M13 & M30 & M32 & M34 & E43 & E44 & E63 & E71,3:FBPSPS
      ;ENDFOLD
      ;FOLD {H}
         VW_MPARA_ACT=P85_D
         Act_P1 = P85
         Act_P2 = P85
         VW(#MPARA,TRUE)
         SPS_FERTIG=FALSE
         TRIGGER WHEN DISTANCE=1 DELAY=0 DO SPS_TRIG(10086) PRIO=-1 UP_TIME_OUT=SPS_TIMEOUT
         TRIGGER WHEN PATH=5 DELAY=-50 DO $B_OUT[11]=(14)
         LIN P85 C_DIS
         $ADVANCE=1
      ;ENDFOLD
   ;ENDFOLD
   ;FOLD KLIN VB=200[mm/s] Genau=40[mm] ACC=50% RobWzg=1 Base=2 SPSTrig=0[1/100s] P ;%{P}%MKUKATPVW,%CMOVE8,%VKLIN,%P 1:4, 2: VB=, 3:200, 4:[mm/s], 5: Genau=, 6:40, 7:[mm], 8: ACC=, 9:50, 10:%, 11: RobWzg=, 12:1, 13: Base=, 14:2, 15: SPSTrig=, 16:0, 17:[1/100s], 18: P, 19:86, 20:-1, 21:87
      ;FOLD 1: FB PSPS = M13 & M30 & M32 & M34 & E43 & E44 & E63 & E71 ;%{SE}%MKUKATPVW %CVW_SPS %VFBPSPS %P 2:FB PSPS = M13 & M30 & M32 & M34 & E43 & E44 & E63 & E71,3:FBPSPS
      ;ENDFOLD
      ;FOLD {H}
         VW_MPARA_ACT=P86_D
         Act_P1 = P86
         Act_P2 = P86
         VW(#MPARA,TRUE)
         SPS_FERTIG=FALSE
         TRIGGER WHEN DISTANCE=1 DELAY=0 DO SPS_TRIG(10087) PRIO=-1 UP_TIME_OUT=SPS_TIMEOUT
         LIN P86 C_DIS
         $ADVANCE=1
      ;ENDFOLD
   ;ENDFOLD
   ;FOLD KLIN VB=200[mm/s] Genau=40[mm] ACC=50% RobWzg=1 Base=2 SPSTrig=0[1/100s] P ;%{P}%MKUKATPVW,%CMOVE8,%VKLIN,%P 1:4, 2: VB=, 3:200, 4:[mm/s], 5: Genau=, 6:40, 7:[mm], 8: ACC=, 9:50, 10:%, 11: RobWzg=, 12:1, 13: Base=, 14:2, 15: SPSTrig=, 16:0, 17:[1/100s], 18: P, 19:87, 20:-1, 21:88
      ;FOLD 1: FB PSPS = M13 & M30 & M32 & M34 & E43 & E44 & E63 & E71 ;%{SE}%MKUKATPVW %CVW_SPS %VFBPSPS %P 2:FB PSPS = M13 & M30 & M32 & M34 & E43 & E44 & E63 & E71,3:FBPSPS
      ;ENDFOLD
      ;FOLD {H}
         VW_MPARA_ACT=P87_D
         Act_P1 = P87
         Act_P2 = P87
         VW(#MPARA,TRUE)
         SPS_FERTIG=FALSE
         TRIGGER WHEN DISTANCE=1 DELAY=0 DO SPS_TRIG(10088) PRIO=-1 UP_TIME_OUT=SPS_TIMEOUT
         LIN P87 C_DIS
         $ADVANCE=1
      ;ENDFOLD
   ;ENDFOLD
   ;FOLD KLIN VB=200[mm/s] Genau=40[mm] ACC=50% RobWzg=1 Base=2 SPSTrig=0[1/100s] P ;%{P}%MKUKATPVW,%CMOVE8,%VKLIN,%P 1:4, 2: VB=, 3:200, 4:[mm/s], 5: Genau=, 6:40, 7:[mm], 8: ACC=, 9:50, 10:%, 11: RobWzg=, 12:1, 13: Base=, 14:2, 15: SPSTrig=, 16:0, 17:[1/100s], 18: P, 19:88, 20:-1, 21:89
      ;FOLD 1: FB PSPS = M13 & M30 & M32 & M34 & E43 & E44 & E63 & E71 ;%{SE}%MKUKATPVW %CVW_SPS %VFBPSPS %P 2:FB PSPS = M13 & M30 & M32 & M34 & E43 & E44 & E63 & E71,3:FBPSPS
      ;ENDFOLD
      ;FOLD {H}
         VW_MPARA_ACT=P88_D
         Act_P1 = P88
         Act_P2 = P88
         VW(#MPARA,TRUE)
         SPS_FERTIG=FALSE
         TRIGGER WHEN DISTANCE=1 DELAY=0 DO SPS_TRIG(10089) PRIO=-1 UP_TIME_OUT=SPS_TIMEOUT
         LIN P88 C_DIS
         $ADVANCE=1
      ;ENDFOLD
   ;ENDFOLD
   ;FOLD -- Schaltpunkt 15 -- ;%{PSE}%MKUKATPVW,%CVW_COM,%VCOMMENT,%P 1:Comment:, 2:Schaltpunkt 15
      ;FOLD {H}
         M_COMMENT("Schaltpunkt 15")
      ;ENDFOLD
   ;ENDFOLD
   ;FOLD KLIN VB=200[mm/s] Genau=40[mm] ACC=50% RobWzg=1 Base=2 SPSTrig=0[1/100s] P ;%{P}%MKUKATPVW,%CMOVE8,%VKLIN,%P 1:4, 2: VB=, 3:200, 4:[mm/s], 5: Genau=, 6:40, 7:[mm], 8: ACC=, 9:50, 10:%, 11: RobWzg=, 12:1, 13: Base=, 14:2, 15: SPSTrig=, 16:0, 17:[1/100s], 18: P, 19:89, 20:-1, 21:90
      ;FOLD BS bin11 ( EIN ) = 15 Schaltpkt:5[mm]:-50[ms] ;%{SE}%MKUKATPVW %CVW_SPS %VBSARI %P 2:BS bin11 ( EIN ) = 15 Schaltpkt:5[mm]:-50[ms],3:BSARI
      ;ENDFOLD
      ;FOLD 1: FB PSPS = M13 & M30 & M32 & M34 & E43 & E44 & E63 & E71 ;%{SE}%MKUKATPVW %CVW_SPS %VFBPSPS %P 2:FB PSPS = M13 & M30 & M32 & M34 & E43 & E44 & E63 & E71,3:FBPSPS
      ;ENDFOLD
      ;FOLD {H}
         VW_MPARA_ACT=P89_D
         Act_P1 = P89
         Act_P2 = P89
         VW(#MPARA,TRUE)
         SPS_FERTIG=FALSE
         TRIGGER WHEN DISTANCE=1 DELAY=0 DO SPS_TRIG(10090) PRIO=-1 UP_TIME_OUT=SPS_TIMEOUT
         TRIGGER WHEN PATH=5 DELAY=-50 DO $B_OUT[11]=(15)
         LIN P89 C_DIS
         $ADVANCE=1
      ;ENDFOLD
   ;ENDFOLD
   ;FOLD KLIN VB=200[mm/s] Genau=40[mm] ACC=50% RobWzg=1 Base=2 SPSTrig=0[1/100s] P ;%{P}%MKUKATPVW,%CMOVE8,%VKLIN,%P 1:4, 2: VB=, 3:200, 4:[mm/s], 5: Genau=, 6:40, 7:[mm], 8: ACC=, 9:50, 10:%, 11: RobWzg=, 12:1, 13: Base=, 14:2, 15: SPSTrig=, 16:0, 17:[1/100s], 18: P, 19:90, 20:-1, 21:91
      ;FOLD 1: FB PSPS = M13 & M30 & M32 & M34 & E43 & E44 & E63 & E71 ;%{SE}%MKUKATPVW %CVW_SPS %VFBPSPS %P 2:FB PSPS = M13 & M30 & M32 & M34 & E43 & E44 & E63 & E71,3:FBPSPS
      ;ENDFOLD
      ;FOLD {H}
         VW_MPARA_ACT=P90_D
         Act_P1 = P90
         Act_P2 = P90
         VW(#MPARA,TRUE)
         SPS_FERTIG=FALSE
         TRIGGER WHEN DISTANCE=1 DELAY=0 DO SPS_TRIG(10091) PRIO=-1 UP_TIME_OUT=SPS_TIMEOUT
         LIN P90 C_DIS
         $ADVANCE=1
      ;ENDFOLD
   ;ENDFOLD
   ;FOLD KLIN VB=200[mm/s] Genau=40[mm] ACC=50% RobWzg=1 Base=2 SPSTrig=0[1/100s] P ;%{P}%MKUKATPVW,%CMOVE8,%VKLIN,%P 1:4, 2: VB=, 3:200, 4:[mm/s], 5: Genau=, 6:40, 7:[mm], 8: ACC=, 9:50, 10:%, 11: RobWzg=, 12:1, 13: Base=, 14:2, 15: SPSTrig=, 16:0, 17:[1/100s], 18: P, 19:91, 20:-1, 21:92
      ;FOLD 1: FB PSPS = M13 & M30 & M32 & M34 & E43 & E44 & E63 & E71 ;%{SE}%MKUKATPVW %CVW_SPS %VFBPSPS %P 2:FB PSPS = M13 & M30 & M32 & M34 & E43 & E44 & E63 & E71,3:FBPSPS
      ;ENDFOLD
      ;FOLD {H}
         VW_MPARA_ACT=P91_D
         Act_P1 = P91
         Act_P2 = P91
         VW(#MPARA,TRUE)
         SPS_FERTIG=FALSE
         TRIGGER WHEN DISTANCE=1 DELAY=0 DO SPS_TRIG(10092) PRIO=-1 UP_TIME_OUT=SPS_TIMEOUT
         LIN P91 C_DIS
         $ADVANCE=1
      ;ENDFOLD
   ;ENDFOLD
   ;FOLD KLIN VB=200[mm/s] Genau=40[mm] ACC=50% RobWzg=1 Base=2 SPSTrig=0[1/100s] P ;%{P}%MKUKATPVW,%CMOVE8,%VKLIN,%P 1:4, 2: VB=, 3:200, 4:[mm/s], 5: Genau=, 6:40, 7:[mm], 8: ACC=, 9:50, 10:%, 11: RobWzg=, 12:1, 13: Base=, 14:2, 15: SPSTrig=, 16:0, 17:[1/100s], 18: P, 19:92, 20:-1, 21:93
      ;FOLD 1: FB PSPS = M13 & M30 & M32 & M34 & E43 & E44 & E63 & E71 ;%{SE}%MKUKATPVW %CVW_SPS %VFBPSPS %P 2:FB PSPS = M13 & M30 & M32 & M34 & E43 & E44 & E63 & E71,3:FBPSPS
      ;ENDFOLD
      ;FOLD {H}
         VW_MPARA_ACT=P92_D
         Act_P1 = P92
         Act_P2 = P92
         VW(#MPARA,TRUE)
         SPS_FERTIG=FALSE
         TRIGGER WHEN DISTANCE=1 DELAY=0 DO SPS_TRIG(10093) PRIO=-1 UP_TIME_OUT=SPS_TIMEOUT
         LIN P92 C_DIS
         $ADVANCE=1
      ;ENDFOLD
   ;ENDFOLD
   ;FOLD KLIN VB=200[mm/s] Genau=40[mm] ACC=50% RobWzg=1 Base=2 SPSTrig=0[1/100s] P ;%{P}%MKUKATPVW,%CMOVE8,%VKLIN,%P 1:4, 2: VB=, 3:200, 4:[mm/s], 5: Genau=, 6:40, 7:[mm], 8: ACC=, 9:50, 10:%, 11: RobWzg=, 12:1, 13: Base=, 14:2, 15: SPSTrig=, 16:0, 17:[1/100s], 18: P, 19:93, 20:-1, 21:94
      ;FOLD 1: FB PSPS = M13 & M30 & M32 & M34 & E43 & E44 & E63 & E71 ;%{SE}%MKUKATPVW %CVW_SPS %VFBPSPS %P 2:FB PSPS = M13 & M30 & M32 & M34 & E43 & E44 & E63 & E71,3:FBPSPS
      ;ENDFOLD
      ;FOLD {H}
         VW_MPARA_ACT=P93_D
         Act_P1 = P93
         Act_P2 = P93
         VW(#MPARA,TRUE)
         SPS_FERTIG=FALSE
         TRIGGER WHEN DISTANCE=1 DELAY=0 DO SPS_TRIG(10094) PRIO=-1 UP_TIME_OUT=SPS_TIMEOUT
         LIN P93 C_DIS
         $ADVANCE=1
      ;ENDFOLD
   ;ENDFOLD
   ;FOLD KLIN VB=200[mm/s] Genau=40[mm] ACC=50% RobWzg=1 Base=2 SPSTrig=0[1/100s] P ;%{P}%MKUKATPVW,%CMOVE8,%VKLIN,%P 1:4, 2: VB=, 3:200, 4:[mm/s], 5: Genau=, 6:40, 7:[mm], 8: ACC=, 9:50, 10:%, 11: RobWzg=, 12:1, 13: Base=, 14:2, 15: SPSTrig=, 16:0, 17:[1/100s], 18: P, 19:94, 20:-1, 21:95
      ;FOLD 1: FB PSPS = M13 & M30 & M32 & M34 & E43 & E44 & E63 & E71 ;%{SE}%MKUKATPVW %CVW_SPS %VFBPSPS %P 2:FB PSPS = M13 & M30 & M32 & M34 & E43 & E44 & E63 & E71,3:FBPSPS
      ;ENDFOLD
      ;FOLD {H}
         VW_MPARA_ACT=P94_D
         Act_P1 = P94
         Act_P2 = P94
         VW(#MPARA,TRUE)
         SPS_FERTIG=FALSE
         TRIGGER WHEN DISTANCE=1 DELAY=0 DO SPS_TRIG(10095) PRIO=-1 UP_TIME_OUT=SPS_TIMEOUT
         LIN P94 C_DIS
         $ADVANCE=1
      ;ENDFOLD
   ;ENDFOLD
   ;FOLD KLIN VB=200[mm/s] Genau=40[mm] ACC=50% RobWzg=1 Base=2 SPSTrig=0[1/100s] P ;%{P}%MKUKATPVW,%CMOVE8,%VKLIN,%P 1:4, 2: VB=, 3:200, 4:[mm/s], 5: Genau=, 6:40, 7:[mm], 8: ACC=, 9:50, 10:%, 11: RobWzg=, 12:1, 13: Base=, 14:2, 15: SPSTrig=, 16:0, 17:[1/100s], 18: P, 19:95, 20:-1, 21:96
      ;FOLD 1: FB PSPS = M13 & M30 & M32 & M34 & E43 & E44 & E63 & E71 ;%{SE}%MKUKATPVW %CVW_SPS %VFBPSPS %P 2:FB PSPS = M13 & M30 & M32 & M34 & E43 & E44 & E63 & E71,3:FBPSPS
      ;ENDFOLD
      ;FOLD {H}
         VW_MPARA_ACT=P95_D
         Act_P1 = P95
         Act_P2 = P95
         VW(#MPARA,TRUE)
         SPS_FERTIG=FALSE
         TRIGGER WHEN DISTANCE=1 DELAY=0 DO SPS_TRIG(10096) PRIO=-1 UP_TIME_OUT=SPS_TIMEOUT
         LIN P95 C_DIS
         $ADVANCE=1
      ;ENDFOLD
   ;ENDFOLD
   ;FOLD KLIN VB=200[mm/s] Genau=40[mm] ACC=50% RobWzg=1 Base=2 SPSTrig=0[1/100s] P ;%{P}%MKUKATPVW,%CMOVE8,%VKLIN,%P 1:4, 2: VB=, 3:200, 4:[mm/s], 5: Genau=, 6:40, 7:[mm], 8: ACC=, 9:50, 10:%, 11: RobWzg=, 12:1, 13: Base=, 14:2, 15: SPSTrig=, 16:0, 17:[1/100s], 18: P, 19:96, 20:-1, 21:97
      ;FOLD 1: FB PSPS = M13 & M30 & M32 & M34 & E43 & E44 & E63 & E71 ;%{SE}%MKUKATPVW %CVW_SPS %VFBPSPS %P 2:FB PSPS = M13 & M30 & M32 & M34 & E43 & E44 & E63 & E71,3:FBPSPS
      ;ENDFOLD
      ;FOLD {H}
         VW_MPARA_ACT=P96_D
         Act_P1 = P96
         Act_P2 = P96
         VW(#MPARA,TRUE)
         SPS_FERTIG=FALSE
         TRIGGER WHEN DISTANCE=1 DELAY=0 DO SPS_TRIG(10097) PRIO=-1 UP_TIME_OUT=SPS_TIMEOUT
         LIN P96 C_DIS
         $ADVANCE=1
      ;ENDFOLD
   ;ENDFOLD
   ;FOLD KLIN VB=200[mm/s] Genau=40[mm] ACC=50% RobWzg=1 Base=2 SPSTrig=0[1/100s] P ;%{P}%MKUKATPVW,%CMOVE8,%VKLIN,%P 1:4, 2: VB=, 3:200, 4:[mm/s], 5: Genau=, 6:40, 7:[mm], 8: ACC=, 9:50, 10:%, 11: RobWzg=, 12:1, 13: Base=, 14:2, 15: SPSTrig=, 16:0, 17:[1/100s], 18: P, 19:97, 20:-1, 21:98
      ;FOLD 1: FB PSPS = M13 & M30 & M32 & M34 & E43 & E44 & E63 & E71 ;%{SE}%MKUKATPVW %CVW_SPS %VFBPSPS %P 2:FB PSPS = M13 & M30 & M32 & M34 & E43 & E44 & E63 & E71,3:FBPSPS
      ;ENDFOLD
      ;FOLD {H}
         VW_MPARA_ACT=P97_D
         Act_P1 = P97
         Act_P2 = P97
         VW(#MPARA,TRUE)
         SPS_FERTIG=FALSE
         TRIGGER WHEN DISTANCE=1 DELAY=0 DO SPS_TRIG(10098) PRIO=-1 UP_TIME_OUT=SPS_TIMEOUT
         LIN P97 C_DIS
         $ADVANCE=1
      ;ENDFOLD
   ;ENDFOLD
   ;FOLD KLIN VB=200[mm/s] Genau=40[mm] ACC=50% RobWzg=1 Base=2 SPSTrig=0[1/100s] P ;%{P}%MKUKATPVW,%CMOVE8,%VKLIN,%P 1:4, 2: VB=, 3:200, 4:[mm/s], 5: Genau=, 6:40, 7:[mm], 8: ACC=, 9:50, 10:%, 11: RobWzg=, 12:1, 13: Base=, 14:2, 15: SPSTrig=, 16:0, 17:[1/100s], 18: P, 19:98, 20:-1, 21:99
      ;FOLD 1: FB PSPS = M13 & M30 & M32 & M34 & E43 & E44 & E63 & E71 ;%{SE}%MKUKATPVW %CVW_SPS %VFBPSPS %P 2:FB PSPS = M13 & M30 & M32 & M34 & E43 & E44 & E63 & E71,3:FBPSPS
      ;ENDFOLD
      ;FOLD {H}
         VW_MPARA_ACT=P98_D
         Act_P1 = P98
         Act_P2 = P98
         VW(#MPARA,TRUE)
         SPS_FERTIG=FALSE
         TRIGGER WHEN DISTANCE=1 DELAY=0 DO SPS_TRIG(10099) PRIO=-1 UP_TIME_OUT=SPS_TIMEOUT
         LIN P98 C_DIS
         $ADVANCE=1
      ;ENDFOLD
   ;ENDFOLD
   ;FOLD KLIN VB=200[mm/s] Genau=40[mm] ACC=50% RobWzg=1 Base=2 SPSTrig=0[1/100s] P ;%{P}%MKUKATPVW,%CMOVE8,%VKLIN,%P 1:4, 2: VB=, 3:200, 4:[mm/s], 5: Genau=, 6:40, 7:[mm], 8: ACC=, 9:50, 10:%, 11: RobWzg=, 12:1, 13: Base=, 14:2, 15: SPSTrig=, 16:0, 17:[1/100s], 18: P, 19:99, 20:-1, 21:100
      ;FOLD 1: FB PSPS = M13 & M30 & M32 & M34 & E43 & E44 & E63 & E71 ;%{SE}%MKUKATPVW %CVW_SPS %VFBPSPS %P 2:FB PSPS = M13 & M30 & M32 & M34 & E43 & E44 & E63 & E71,3:FBPSPS
      ;ENDFOLD
      ;FOLD {H}
         VW_MPARA_ACT=P99_D
         Act_P1 = P99
         Act_P2 = P99
         VW(#MPARA,TRUE)
         SPS_FERTIG=FALSE
         TRIGGER WHEN DISTANCE=1 DELAY=0 DO SPS_TRIG(10100) PRIO=-1 UP_TIME_OUT=SPS_TIMEOUT
         LIN P99 C_DIS
         $ADVANCE=1
      ;ENDFOLD
   ;ENDFOLD
   ;FOLD KLIN VB=200[mm/s] Genau=40[mm] ACC=50% RobWzg=1 Base=2 SPSTrig=0[1/100s] P ;%{P}%MKUKATPVW,%CMOVE8,%VKLIN,%P 1:4, 2: VB=, 3:200, 4:[mm/s], 5: Genau=, 6:40, 7:[mm], 8: ACC=, 9:50, 10:%, 11: RobWzg=, 12:1, 13: Base=, 14:2, 15: SPSTrig=, 16:0, 17:[1/100s], 18: P, 19:100, 20:-1, 21:101
      ;FOLD 1: FB PSPS = M13 & M30 & M32 & M34 & E43 & E44 & E63 & E71 ;%{SE}%MKUKATPVW %CVW_SPS %VFBPSPS %P 2:FB PSPS = M13 & M30 & M32 & M34 & E43 & E44 & E63 & E71,3:FBPSPS
      ;ENDFOLD
      ;FOLD {H}
         VW_MPARA_ACT=P100_D
         Act_P1 = P100
         Act_P2 = P100
         VW(#MPARA,TRUE)
         SPS_FERTIG=FALSE
         TRIGGER WHEN DISTANCE=1 DELAY=0 DO SPS_TRIG(10101) PRIO=-1 UP_TIME_OUT=SPS_TIMEOUT
         LIN P100 C_DIS
         $ADVANCE=1
      ;ENDFOLD
   ;ENDFOLD
   ;FOLD KLIN VB=200[mm/s] Genau=40[mm] ACC=50% RobWzg=1 Base=2 SPSTrig=0[1/100s] P ;%{P}%MKUKATPVW,%CMOVE8,%VKLIN,%P 1:4, 2: VB=, 3:200, 4:[mm/s], 5: Genau=, 6:40, 7:[mm], 8: ACC=, 9:50, 10:%, 11: RobWzg=, 12:1, 13: Base=, 14:2, 15: SPSTrig=, 16:0, 17:[1/100s], 18: P, 19:101, 20:-1, 21:102
      ;FOLD 1: FB PSPS = M13 & M30 & M32 & M34 & E43 & E44 & E63 & E71 ;%{SE}%MKUKATPVW %CVW_SPS %VFBPSPS %P 2:FB PSPS = M13 & M30 & M32 & M34 & E43 & E44 & E63 & E71,3:FBPSPS
      ;ENDFOLD
      ;FOLD {H}
         VW_MPARA_ACT=P101_D
         Act_P1 = P101
         Act_P2 = P101
         VW(#MPARA,TRUE)
         SPS_FERTIG=FALSE
         TRIGGER WHEN DISTANCE=1 DELAY=0 DO SPS_TRIG(10102) PRIO=-1 UP_TIME_OUT=SPS_TIMEOUT
         LIN P101 C_DIS
         $ADVANCE=1
      ;ENDFOLD
   ;ENDFOLD
   ;FOLD -- Schaltpunkt 16 -- ;%{PSE}%MKUKATPVW,%CVW_COM,%VCOMMENT,%P 1:Comment:, 2:Schaltpunkt 16
      ;FOLD {H}
         M_COMMENT("Schaltpunkt 16")
      ;ENDFOLD
   ;ENDFOLD
   ;FOLD KLIN VB=200[mm/s] Genau=40[mm] ACC=50% RobWzg=1 Base=2 SPSTrig=0[1/100s] P ;%{P}%MKUKATPVW,%CMOVE8,%VKLIN,%P 1:4, 2: VB=, 3:200, 4:[mm/s], 5: Genau=, 6:40, 7:[mm], 8: ACC=, 9:50, 10:%, 11: RobWzg=, 12:1, 13: Base=, 14:2, 15: SPSTrig=, 16:0, 17:[1/100s], 18: P, 19:102, 20:-1, 21:103
      ;FOLD BS bin11 ( EIN ) = 16 Schaltpkt:5[mm]:-50[ms] ;%{SE}%MKUKATPVW %CVW_SPS %VBSARI %P 2:BS bin11 ( EIN ) = 16 Schaltpkt:5[mm]:-50[ms],3:BSARI
      ;ENDFOLD
      ;FOLD 1: FB PSPS = M13 & M30 & M32 & M34 & E43 & E44 & E63 & E71 ;%{SE}%MKUKATPVW %CVW_SPS %VFBPSPS %P 2:FB PSPS = M13 & M30 & M32 & M34 & E43 & E44 & E63 & E71,3:FBPSPS
      ;ENDFOLD
      ;FOLD {H}
         VW_MPARA_ACT=P102_D
         Act_P1 = P102
         Act_P2 = P102
         VW(#MPARA,TRUE)
         SPS_FERTIG=FALSE
         TRIGGER WHEN DISTANCE=1 DELAY=0 DO SPS_TRIG(10103) PRIO=-1 UP_TIME_OUT=SPS_TIMEOUT
         TRIGGER WHEN PATH=5 DELAY=-50 DO $B_OUT[11]=(16)
         LIN P102 C_DIS
         $ADVANCE=1
      ;ENDFOLD
   ;ENDFOLD
   ;FOLD KLIN VB=200[mm/s] Genau=40[mm] ACC=50% RobWzg=1 Base=2 SPSTrig=0[1/100s] P ;%{P}%MKUKATPVW,%CMOVE8,%VKLIN,%P 1:4, 2: VB=, 3:200, 4:[mm/s], 5: Genau=, 6:40, 7:[mm], 8: ACC=, 9:50, 10:%, 11: RobWzg=, 12:1, 13: Base=, 14:2, 15: SPSTrig=, 16:0, 17:[1/100s], 18: P, 19:103, 20:-1, 21:104
      ;FOLD 1: FB PSPS = M13 & M30 & M32 & M34 & E43 & E44 & E63 & E71 ;%{SE}%MKUKATPVW %CVW_SPS %VFBPSPS %P 2:FB PSPS = M13 & M30 & M32 & M34 & E43 & E44 & E63 & E71,3:FBPSPS
      ;ENDFOLD
      ;FOLD {H}
         VW_MPARA_ACT=P103_D
         Act_P1 = P103
         Act_P2 = P103
         VW(#MPARA,TRUE)
         SPS_FERTIG=FALSE
         TRIGGER WHEN DISTANCE=1 DELAY=0 DO SPS_TRIG(10104) PRIO=-1 UP_TIME_OUT=SPS_TIMEOUT
         LIN P103 C_DIS
         $ADVANCE=1
      ;ENDFOLD
   ;ENDFOLD
   ;FOLD KLIN VB=200[mm/s] Genau=40[mm] ACC=50% RobWzg=1 Base=2 SPSTrig=0[1/100s] P ;%{P}%MKUKATPVW,%CMOVE8,%VKLIN,%P 1:4, 2: VB=, 3:200, 4:[mm/s], 5: Genau=, 6:40, 7:[mm], 8: ACC=, 9:50, 10:%, 11: RobWzg=, 12:1, 13: Base=, 14:2, 15: SPSTrig=, 16:0, 17:[1/100s], 18: P, 19:104, 20:-1, 21:105
      ;FOLD 1: FB PSPS = M13 & M30 & M32 & M34 & E43 & E44 & E63 & E71 ;%{SE}%MKUKATPVW %CVW_SPS %VFBPSPS %P 2:FB PSPS = M13 & M30 & M32 & M34 & E43 & E44 & E63 & E71,3:FBPSPS
      ;ENDFOLD
      ;FOLD {H}
         VW_MPARA_ACT=P104_D
         Act_P1 = P104
         Act_P2 = P104
         VW(#MPARA,TRUE)
         SPS_FERTIG=FALSE
         TRIGGER WHEN DISTANCE=1 DELAY=0 DO SPS_TRIG(10105) PRIO=-1 UP_TIME_OUT=SPS_TIMEOUT
         LIN P104 C_DIS
         $ADVANCE=1
      ;ENDFOLD
   ;ENDFOLD
   ;FOLD KLIN VB=200[mm/s] Genau=40[mm] ACC=50% RobWzg=1 Base=2 SPSTrig=0[1/100s] P ;%{P}%MKUKATPVW,%CMOVE8,%VKLIN,%P 1:4, 2: VB=, 3:200, 4:[mm/s], 5: Genau=, 6:40, 7:[mm], 8: ACC=, 9:50, 10:%, 11: RobWzg=, 12:1, 13: Base=, 14:2, 15: SPSTrig=, 16:0, 17:[1/100s], 18: P, 19:105, 20:-1, 21:106
      ;FOLD 1: FB PSPS = M13 & M30 & M32 & M34 & E43 & E44 & E63 & E71 ;%{SE}%MKUKATPVW %CVW_SPS %VFBPSPS %P 2:FB PSPS = M13 & M30 & M32 & M34 & E43 & E44 & E63 & E71,3:FBPSPS
      ;ENDFOLD
      ;FOLD {H}
         VW_MPARA_ACT=P105_D
         Act_P1 = P105
         Act_P2 = P105
         VW(#MPARA,TRUE)
         SPS_FERTIG=FALSE
         TRIGGER WHEN DISTANCE=1 DELAY=0 DO SPS_TRIG(10106) PRIO=-1 UP_TIME_OUT=SPS_TIMEOUT
         LIN P105 C_DIS
         $ADVANCE=1
      ;ENDFOLD
   ;ENDFOLD
   ;FOLD KLIN VB=200[mm/s] Genau=40[mm] ACC=50% RobWzg=1 Base=2 SPSTrig=0[1/100s] P ;%{P}%MKUKATPVW,%CMOVE8,%VKLIN,%P 1:4, 2: VB=, 3:200, 4:[mm/s], 5: Genau=, 6:40, 7:[mm], 8: ACC=, 9:50, 10:%, 11: RobWzg=, 12:1, 13: Base=, 14:2, 15: SPSTrig=, 16:0, 17:[1/100s], 18: P, 19:106, 20:-1, 21:107
